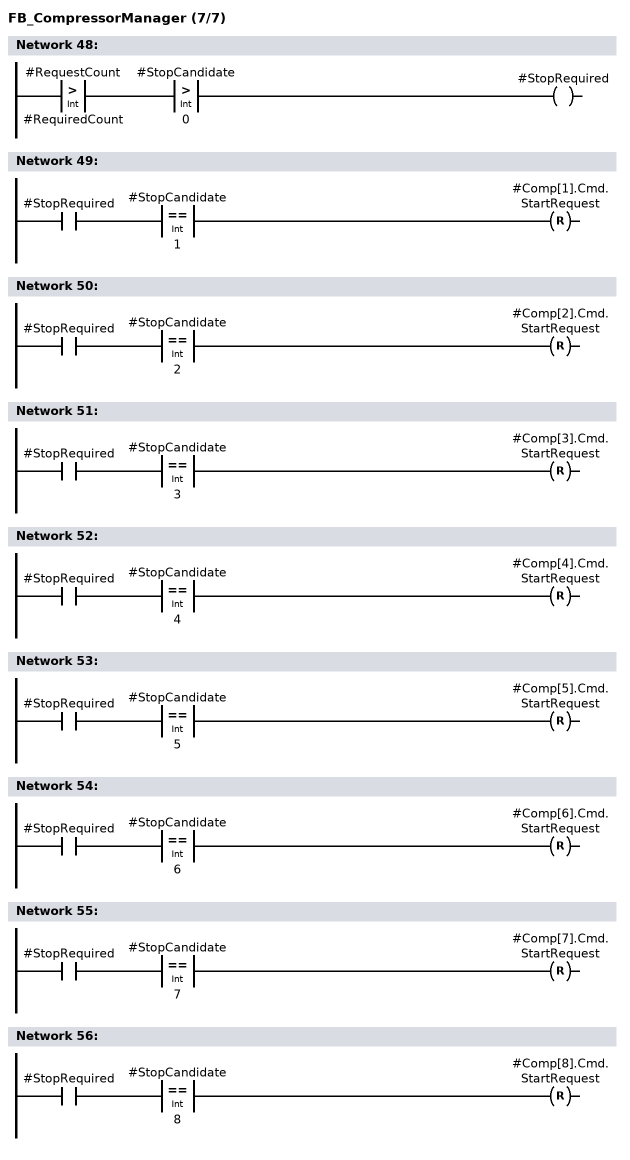
   RUNG wire#powerrail
      { S7_Templates := "SrcType := Int" } GT_Contact(in1 := #RequestCount, in2 := #RequiredCount)
      { S7_Templates := "SrcType := Int" } GT_Contact(in1 := #StopCandidate, in2 := 0)
      Coil( #StopRequired )
   END_RUNG
   // the same network as SCL:
   #StopRequired := (#RequestCount > #RequiredCount) AND (#StopCandidate > 0);
END_REGION

REGION Network 49
   RUNG wire#powerrail
      Contact( #StopRequired )
      { S7_Templates := "SrcType := Int" } EQ_Contact(in1 := #StopCandidate, in2 := 1)
      R_Coil( #Comp[1].Cmd.StartRequest )
   END_RUNG
   // the same network as SCL:
   IF #StopRequired AND (#StopCandidate = 1) THEN #Comp[1].Cmd.StartRequest := FALSE; END_IF;
END_REGION

REGION Network 50
   RUNG wire#powerrail
      Contact( #StopRequired )
      { S7_Templates := "SrcType := Int" } EQ_Contact(in1 := #StopCandidate, in2 := 2)
      R_Coil( #Comp[2].Cmd.StartRequest )
   END_RUNG
   // the same network as SCL:
   IF #StopRequired AND (#StopCandidate = 2) THEN #Comp[2].Cmd.StartRequest := FALSE; END_IF;
END_REGION

REGION Network 51
   RUNG wire#powerrail
      Contact( #StopRequired )
      { S7_Templates := "SrcType := Int" } EQ_Contact(in1 := #StopCandidate, in2 := 3)
      R_Coil( #Comp[3].Cmd.StartRequest )
   END_RUNG
   // the same network as SCL:
   IF #StopRequired AND (#StopCandidate = 3) THEN #Comp[3].Cmd.StartRequest := FALSE; END_IF;
END_REGION

REGION Network 52
   RUNG wire#powerrail
      Contact( #StopRequired )
      { S7_Templates := "SrcType := Int" } EQ_Contact(in1 := #StopCandidate, in2 := 4)
      R_Coil( #Comp[4].Cmd.StartRequest )
   END_RUNG
   // the same network as SCL:
   IF #StopRequired AND (#StopCandidate = 4) THEN #Comp[4].Cmd.StartRequest := FALSE; END_IF;
END_REGION

REGION Network 53
   RUNG wire#powerrail
      Contact( #StopRequired )
      { S7_Templates := "SrcType := Int" } EQ_Contact(in1 := #StopCandidate, in2 := 5)
      R_Coil( #Comp[5].Cmd.StartRequest )
   END_RUNG
   // the same network as SCL:
   IF #StopRequired AND (#StopCandidate = 5) THEN #Comp[5].Cmd.StartRequest := FALSE; END_IF;
END_REGION

REGION Network 54
   RUNG wire#powerrail
      Contact( #StopRequired )
      { S7_Templates := "SrcType := Int" } EQ_Contact(in1 := #StopCandidate, in2 := 6)
      R_Coil( #Comp[6].Cmd.StartRequest )
   END_RUNG
   // the same network as SCL:
   IF #StopRequired AND (#StopCandidate = 6) THEN #Comp[6].Cmd.StartRequest := FALSE; END_IF;
END_REGION

REGION Network 55
   RUNG wire#powerrail
      Contact( #StopRequired )
      { S7_Templates := "SrcType := Int" } EQ_Contact(in1 := #StopCandidate, in2 := 7)
      R_Coil( #Comp[7].Cmd.StartRequest )
   END_RUNG
   // the same network as SCL:
   IF #StopRequired AND (#StopCandidate = 7) THEN #Comp[7].Cmd.StartRequest := FALSE; END_IF;
END_REGION

REGION Network 56
   RUNG wire#powerrail
      Contact( #StopRequired )
      { S7_Templates := "SrcType := Int" } EQ_Contact(in1 := #StopCandidate, in2 := 8)
      R_Coil( #Comp[8].Cmd.StartRequest )
   END_RUNG
   // the same network as SCL:
   IF #StopRequired AND (#StopCandidate = 8) THEN #Comp[8].Cmd.StartRequest := FALSE; END_IF;
END_REGION
END_FUNCTION_BLOCK

FUNCTION_BLOCK "FB_Fan"   // FB3, LAD
{ S7_Optimized_Access := 'TRUE' }
VERSION : 0.1
   VAR_INPUT
      Timing : "UDT_TimingParams";
   END_VAR
   VAR_IN_OUT
      Fan : "UDT_Fan";
   END_VAR
   VAR
      tMinOff : TON_TIME;
      tMinOn : TON_TIME;
      StartLatch : Bool;
      tFeedBack : TON_TIME;
   END_VAR
   VAR_TEMP
      MinOffDone : Bool;
      MinOnDone : Bool;
      StopCondition : Bool;
      FeedbackTimeOut : Bool;
   END_VAR
BEGIN

REGION Network 1
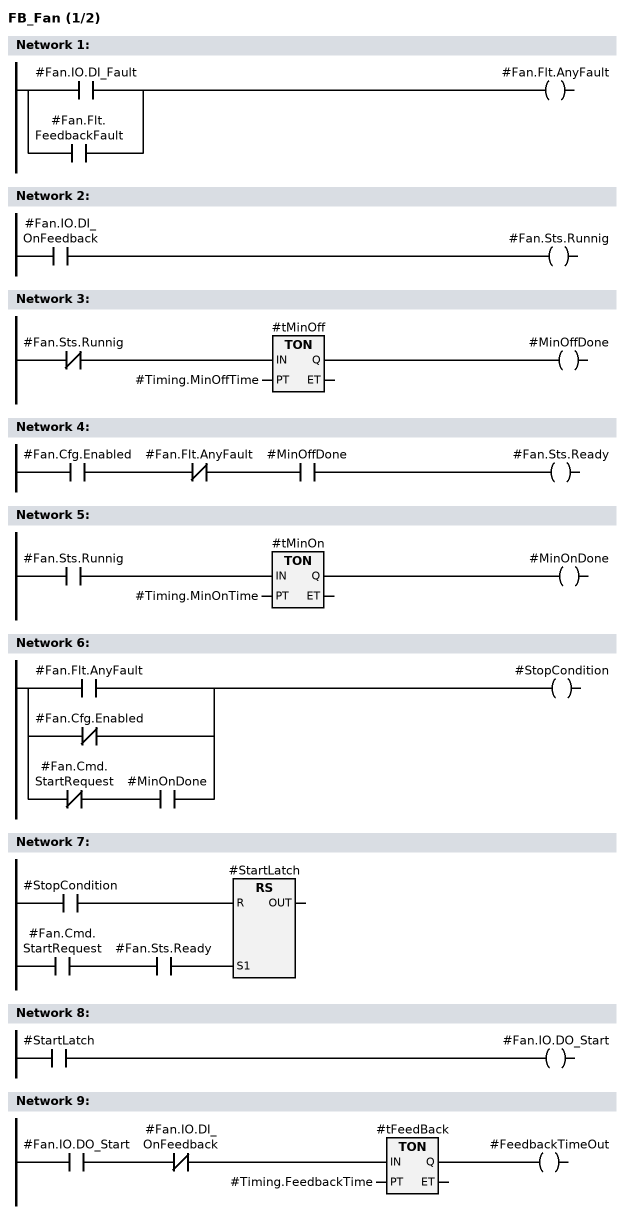
   RUNG wire#powerrail
      Contact( #Fan.IO.DI_Fault )
      wire#w1
      Coil( #Fan.Flt.AnyFault )
   END_RUNG
   RUNG wire#powerrail
      Contact( #Fan.Flt.FeedbackFault )
   END_RUNG wire#w1
   // the same network as SCL:
   #Fan.Flt.AnyFault := #Fan.IO.DI_Fault OR #Fan.Flt.FeedbackFault;
END_REGION

REGION Network 2
   RUNG wire#powerrail
      Contact( #Fan.IO.DI_OnFeedback )
      Coil( #Fan.Sts.Runnig )
   END_RUNG
   // the same network as SCL:
   #Fan.Sts.Runnig := #Fan.IO.DI_OnFeedback;
END_REGION

REGION Network 3
   #tMinOff(IN := NOT #Fan.Sts.Runnig, PT := #Timing.MinOffTime);   // TON
   #MinOffDone := #tMinOff.Q;
END_REGION

REGION Network 4
   RUNG wire#powerrail
      Contact( #Fan.Cfg.Enabled )
      I_Contact( #Fan.Flt.AnyFault )
      Contact( #MinOffDone )
      Coil( #Fan.Sts.Ready )
   END_RUNG
   // the same network as SCL:
   #Fan.Sts.Ready := #Fan.Cfg.Enabled AND NOT #Fan.Flt.AnyFault AND #MinOffDone;
END_REGION

REGION Network 5
   #tMinOn(IN := #Fan.Sts.Runnig, PT := #Timing.MinOnTime);   // TON
   #MinOnDone := #tMinOn.Q;
END_REGION

REGION Network 6
   RUNG wire#powerrail
      Contact( #Fan.Flt.AnyFault )
      wire#w1
      Coil( #StopCondition )
   END_RUNG
   RUNG wire#powerrail
      I_Contact( #Fan.Cfg.Enabled )
   END_RUNG wire#w1
   RUNG wire#powerrail
      I_Contact( #Fan.Cmd.StartRequest )
      Contact( #MinOnDone )
   END_RUNG wire#w1
   // the same network as SCL:
   #StopCondition := #Fan.Flt.AnyFault OR NOT #Fan.Cfg.Enabled OR (NOT #Fan.Cmd.StartRequest AND #MinOnDone);
END_REGION

REGION Network 7
   RUNG wire#powerrail
      Contact( #StopCondition )
      S_RS(operand := #StartLatch, s1 := wire#w1)
   END_RUNG
   RUNG wire#powerrail
      Contact( #Fan.Cmd.StartRequest )
      Contact( #Fan.Sts.Ready )
   END_RUNG wire#w1
   // the same network as SCL:
   IF #StopCondition THEN
       #StartLatch := FALSE;   // RS flip-flop
   END_IF;
   IF #Fan.Cmd.StartRequest AND #Fan.Sts.Ready THEN #StartLatch := TRUE; END_IF;
END_REGION

REGION Network 8
   RUNG wire#powerrail
      Contact( #StartLatch )
      Coil( #Fan.IO.DO_Start )
   END_RUNG
   // the same network as SCL:
   #Fan.IO.DO_Start := #StartLatch;
END_REGION

REGION Network 9
   #tFeedBack(IN := #Fan.IO.DO_Start AND NOT #Fan.IO.DI_OnFeedback, PT := #Timing.FeedbackTime);   // TON
   #FeedbackTimeOut := #tFeedBack.Q;
END_REGION

REGION Network 10
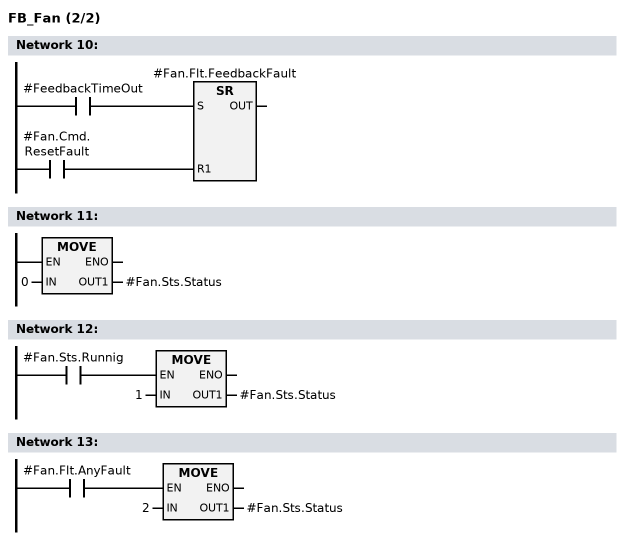
   RUNG wire#powerrail
      Contact( #FeedbackTimeOut )
      S_SR(operand := #Fan.Flt.FeedbackFault, r1 := wire#w1)
   END_RUNG
   RUNG wire#powerrail
      Contact( #Fan.Cmd.ResetFault )
   END_RUNG wire#w1
   // the same network as SCL:
   IF #FeedbackTimeOut THEN
       #Fan.Flt.FeedbackFault := TRUE;   // SR flip-flop
   END_IF;
   IF #Fan.Cmd.ResetFault THEN #Fan.Flt.FeedbackFault := FALSE; END_IF;
END_REGION

REGION Network 11
   RUNG wire#powerrail
      Move(in := 0, out1 => #Fan.Sts.Status)
   END_RUNG
   // the same network as SCL:
   #Fan.Sts.Status := 0;
END_REGION

REGION Network 12
   RUNG wire#powerrail
      Contact( #Fan.Sts.Runnig )
      Move(in := 1, out1 => #Fan.Sts.Status)
   END_RUNG
   // the same network as SCL:
   IF #Fan.Sts.Runnig THEN #Fan.Sts.Status := 1; END_IF;
END_REGION

REGION Network 13
   RUNG wire#powerrail
      Contact( #Fan.Flt.AnyFault )
      Move(in := 2, out1 => #Fan.Sts.Status)
   END_RUNG
   // the same network as SCL:
   IF #Fan.Flt.AnyFault THEN #Fan.Sts.Status := 2; END_IF;
END_REGION
END_FUNCTION_BLOCK

FUNCTION_BLOCK "FB_FanManager"   // FB4, LAD
{ S7_Optimized_Access := 'TRUE' }
VERSION : 0.1
   VAR_INPUT
      Enable : Bool;
      RequiredCount : Int;
   END_VAR
   VAR_OUTPUT
      RunningCount : Int;
      RequestCount : Int;
   END_VAR
   VAR_IN_OUT
      fan : Array[1..12] of "UDT_Fan";
   END_VAR
   VAR_TEMP
      TargetCount : Int;
      StartCandidate : Int;
      StopCandidate : Int;
      StartRequired : Bool;
      StopRequired : Bool;
   END_VAR
BEGIN

REGION Network 1
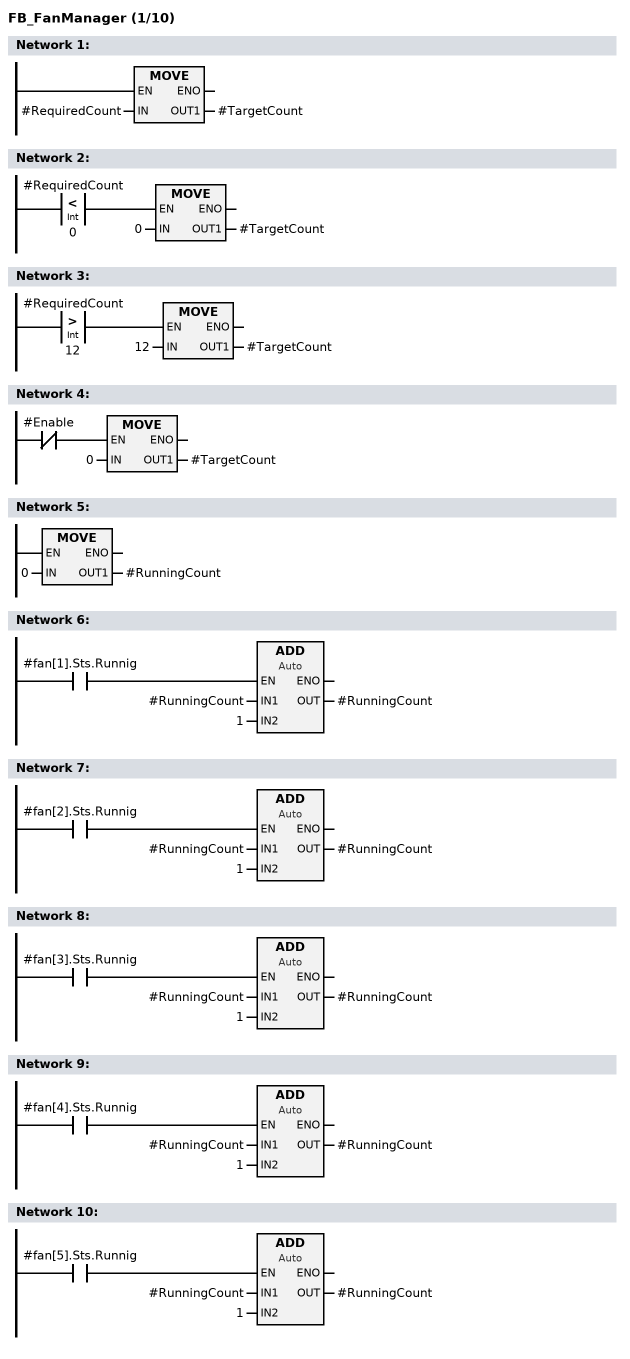
   RUNG wire#powerrail
      Move(in := #RequiredCount, out1 => #TargetCount)
   END_RUNG
   // the same network as SCL:
   #TargetCount := #RequiredCount;
END_REGION

REGION Network 2
   RUNG wire#powerrail
      { S7_Templates := "SrcType := Int" } LT_Contact(in1 := #RequiredCount, in2 := 0)
      Move(in := 0, out1 => #TargetCount)
   END_RUNG
   // the same network as SCL:
   IF #RequiredCount < 0 THEN #TargetCount := 0; END_IF;
END_REGION

REGION Network 3
   RUNG wire#powerrail
      { S7_Templates := "SrcType := Int" } GT_Contact(in1 := #RequiredCount, in2 := 12)
      Move(in := 12, out1 => #TargetCount)
   END_RUNG
   // the same network as SCL:
   IF #RequiredCount > 12 THEN #TargetCount := 12; END_IF;
END_REGION

REGION Network 4
   RUNG wire#powerrail
      I_Contact( #Enable )
      Move(in := 0, out1 => #TargetCount)
   END_RUNG
   // the same network as SCL:
   IF NOT #Enable THEN #TargetCount := 0; END_IF;
END_REGION

REGION Network 5
   RUNG wire#powerrail
      Move(in := 0, out1 => #RunningCount)
   END_RUNG
   // the same network as SCL:
   #RunningCount := 0;
END_REGION

REGION Network 6
   RUNG wire#powerrail
      Contact( #fan[1].Sts.Runnig )
      Add(in1 := #RunningCount, in2 := 1, out => #RunningCount)
   END_RUNG
   // the same network as SCL:
   IF #fan[1].Sts.Runnig THEN #RunningCount := #RunningCount + 1; END_IF;
END_REGION

REGION Network 7
   RUNG wire#powerrail
      Contact( #fan[2].Sts.Runnig )
      Add(in1 := #RunningCount, in2 := 1, out => #RunningCount)
   END_RUNG
   // the same network as SCL:
   IF #fan[2].Sts.Runnig THEN #RunningCount := #RunningCount + 1; END_IF;
END_REGION

REGION Network 8
   RUNG wire#powerrail
      Contact( #fan[3].Sts.Runnig )
      Add(in1 := #RunningCount, in2 := 1, out => #RunningCount)
   END_RUNG
   // the same network as SCL:
   IF #fan[3].Sts.Runnig THEN #RunningCount := #RunningCount + 1; END_IF;
END_REGION

REGION Network 9
   RUNG wire#powerrail
      Contact( #fan[4].Sts.Runnig )
      Add(in1 := #RunningCount, in2 := 1, out => #RunningCount)
   END_RUNG
   // the same network as SCL:
   IF #fan[4].Sts.Runnig THEN #RunningCount := #RunningCount + 1; END_IF;
END_REGION

REGION Network 10
   RUNG wire#powerrail
      Contact( #fan[5].Sts.Runnig )
      Add(in1 := #RunningCount, in2 := 1, out => #RunningCount)
   END_RUNG
   // the same network as SCL:
   IF #fan[5].Sts.Runnig THEN #RunningCount := #RunningCount + 1; END_IF;
END_REGION

REGION Network 11
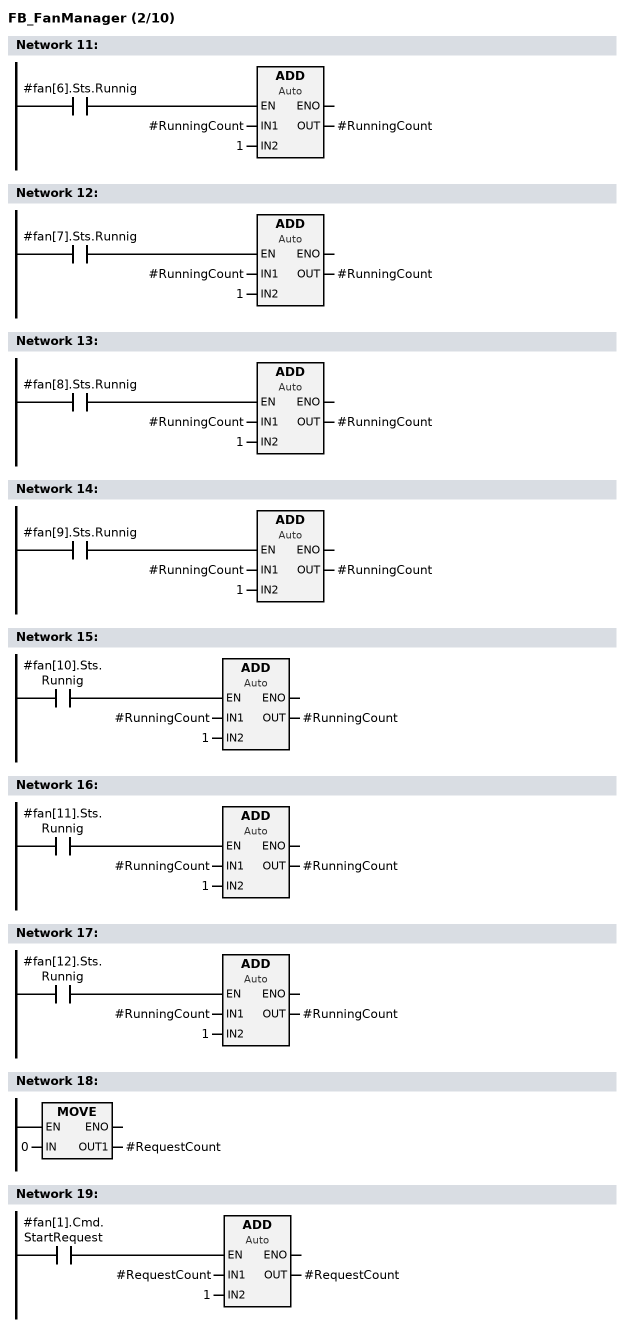
   RUNG wire#powerrail
      Contact( #fan[6].Sts.Runnig )
      Add(in1 := #RunningCount, in2 := 1, out => #RunningCount)
   END_RUNG
   // the same network as SCL:
   IF #fan[6].Sts.Runnig THEN #RunningCount := #RunningCount + 1; END_IF;
END_REGION

REGION Network 12
   RUNG wire#powerrail
      Contact( #fan[7].Sts.Runnig )
      Add(in1 := #RunningCount, in2 := 1, out => #RunningCount)
   END_RUNG
   // the same network as SCL:
   IF #fan[7].Sts.Runnig THEN #RunningCount := #RunningCount + 1; END_IF;
END_REGION

REGION Network 13
   RUNG wire#powerrail
      Contact( #fan[8].Sts.Runnig )
      Add(in1 := #RunningCount, in2 := 1, out => #RunningCount)
   END_RUNG
   // the same network as SCL:
   IF #fan[8].Sts.Runnig THEN #RunningCount := #RunningCount + 1; END_IF;
END_REGION

REGION Network 14
   RUNG wire#powerrail
      Contact( #fan[9].Sts.Runnig )
      Add(in1 := #RunningCount, in2 := 1, out => #RunningCount)
   END_RUNG
   // the same network as SCL:
   IF #fan[9].Sts.Runnig THEN #RunningCount := #RunningCount + 1; END_IF;
END_REGION

REGION Network 15
   RUNG wire#powerrail
      Contact( #fan[10].Sts.Runnig )
      Add(in1 := #RunningCount, in2 := 1, out => #RunningCount)
   END_RUNG
   // the same network as SCL:
   IF #fan[10].Sts.Runnig THEN #RunningCount := #RunningCount + 1; END_IF;
END_REGION

REGION Network 16
   RUNG wire#powerrail
      Contact( #fan[11].Sts.Runnig )
      Add(in1 := #RunningCount, in2 := 1, out => #RunningCount)
   END_RUNG
   // the same network as SCL:
   IF #fan[11].Sts.Runnig THEN #RunningCount := #RunningCount + 1; END_IF;
END_REGION

REGION Network 17
   RUNG wire#powerrail
      Contact( #fan[12].Sts.Runnig )
      Add(in1 := #RunningCount, in2 := 1, out => #RunningCount)
   END_RUNG
   // the same network as SCL:
   IF #fan[12].Sts.Runnig THEN #RunningCount := #RunningCount + 1; END_IF;
END_REGION

REGION Network 18
   RUNG wire#powerrail
      Move(in := 0, out1 => #RequestCount)
   END_RUNG
   // the same network as SCL:
   #RequestCount := 0;
END_REGION

REGION Network 19
   RUNG wire#powerrail
      Contact( #fan[1].Cmd.StartRequest )
      Add(in1 := #RequestCount, in2 := 1, out => #RequestCount)
   END_RUNG
   // the same network as SCL:
   IF #fan[1].Cmd.StartRequest THEN #RequestCount := #RequestCount + 1; END_IF;
END_REGION

REGION Network 20
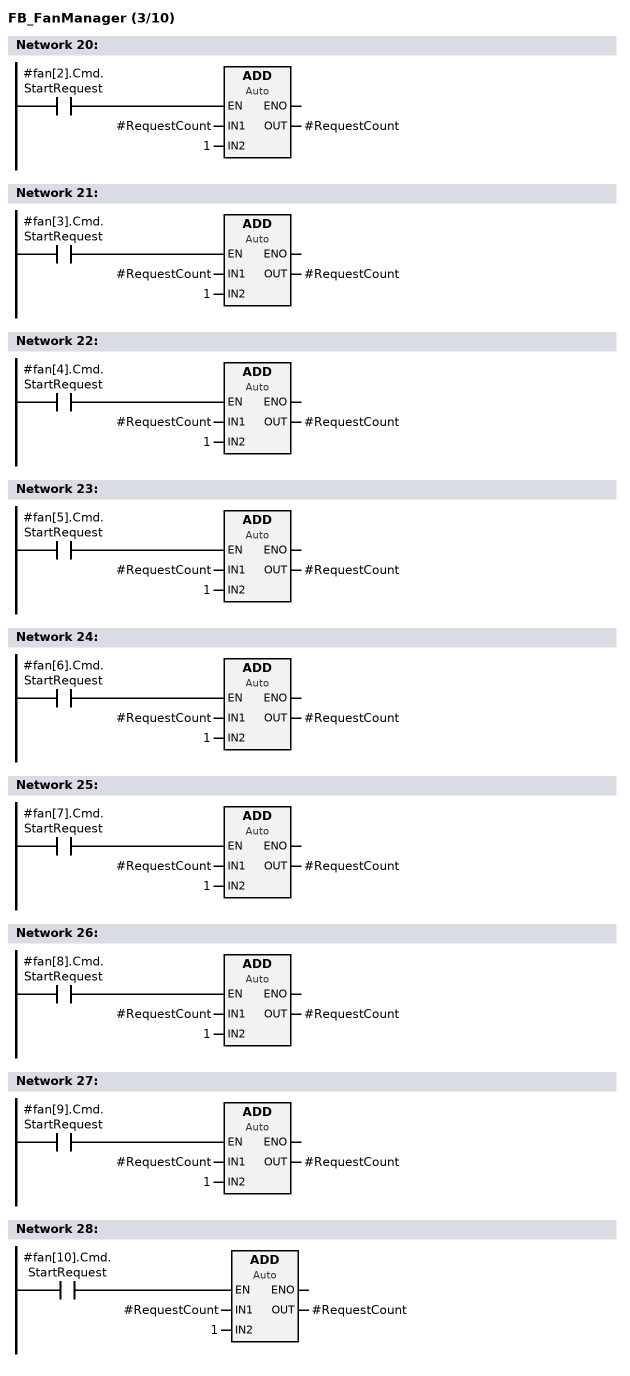
   RUNG wire#powerrail
      Contact( #fan[2].Cmd.StartRequest )
      Add(in1 := #RequestCount, in2 := 1, out => #RequestCount)
   END_RUNG
   // the same network as SCL:
   IF #fan[2].Cmd.StartRequest THEN #RequestCount := #RequestCount + 1; END_IF;
END_REGION

REGION Network 21
   RUNG wire#powerrail
      Contact( #fan[3].Cmd.StartRequest )
      Add(in1 := #RequestCount, in2 := 1, out => #RequestCount)
   END_RUNG
   // the same network as SCL:
   IF #fan[3].Cmd.StartRequest THEN #RequestCount := #RequestCount + 1; END_IF;
END_REGION

REGION Network 22
   RUNG wire#powerrail
      Contact( #fan[4].Cmd.StartRequest )
      Add(in1 := #RequestCount, in2 := 1, out => #RequestCount)
   END_RUNG
   // the same network as SCL:
   IF #fan[4].Cmd.StartRequest THEN #RequestCount := #RequestCount + 1; END_IF;
END_REGION

REGION Network 23
   RUNG wire#powerrail
      Contact( #fan[5].Cmd.StartRequest )
      Add(in1 := #RequestCount, in2 := 1, out => #RequestCount)
   END_RUNG
   // the same network as SCL:
   IF #fan[5].Cmd.StartRequest THEN #RequestCount := #RequestCount + 1; END_IF;
END_REGION

REGION Network 24
   RUNG wire#powerrail
      Contact( #fan[6].Cmd.StartRequest )
      Add(in1 := #RequestCount, in2 := 1, out => #RequestCount)
   END_RUNG
   // the same network as SCL:
   IF #fan[6].Cmd.StartRequest THEN #RequestCount := #RequestCount + 1; END_IF;
END_REGION

REGION Network 25
   RUNG wire#powerrail
      Contact( #fan[7].Cmd.StartRequest )
      Add(in1 := #RequestCount, in2 := 1, out => #RequestCount)
   END_RUNG
   // the same network as SCL:
   IF #fan[7].Cmd.StartRequest THEN #RequestCount := #RequestCount + 1; END_IF;
END_REGION

REGION Network 26
   RUNG wire#powerrail
      Contact( #fan[8].Cmd.StartRequest )
      Add(in1 := #RequestCount, in2 := 1, out => #RequestCount)
   END_RUNG
   // the same network as SCL:
   IF #fan[8].Cmd.StartRequest THEN #RequestCount := #RequestCount + 1; END_IF;
END_REGION

REGION Network 27
   RUNG wire#powerrail
      Contact( #fan[9].Cmd.StartRequest )
      Add(in1 := #RequestCount, in2 := 1, out => #RequestCount)
   END_RUNG
   // the same network as SCL:
   IF #fan[9].Cmd.StartRequest THEN #RequestCount := #RequestCount + 1; END_IF;
END_REGION

REGION Network 28
   RUNG wire#powerrail
      Contact( #fan[10].Cmd.StartRequest )
      Add(in1 := #RequestCount, in2 := 1, out => #RequestCount)
   END_RUNG
   // the same network as SCL:
   IF #fan[10].Cmd.StartRequest THEN #RequestCount := #RequestCount + 1; END_IF;
END_REGION

REGION Network 29
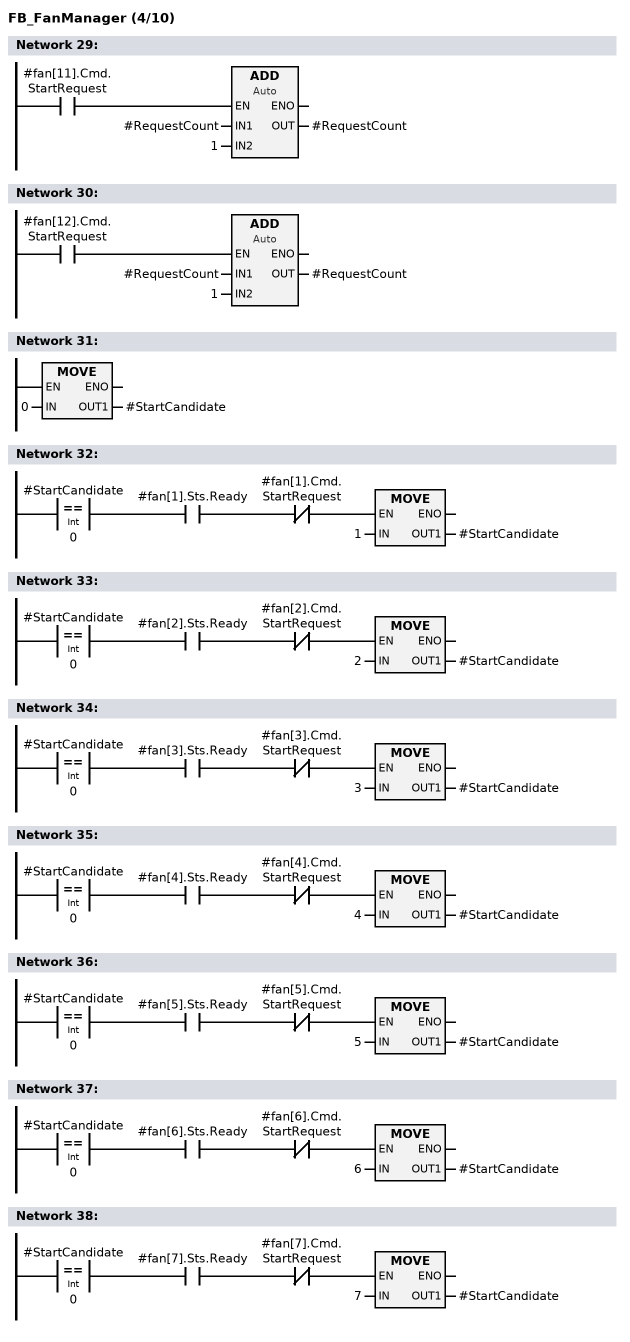
   RUNG wire#powerrail
      Contact( #fan[11].Cmd.StartRequest )
      Add(in1 := #RequestCount, in2 := 1, out => #RequestCount)
   END_RUNG
   // the same network as SCL:
   IF #fan[11].Cmd.StartRequest THEN #RequestCount := #RequestCount + 1; END_IF;
END_REGION

REGION Network 30
   RUNG wire#powerrail
      Contact( #fan[12].Cmd.StartRequest )
      Add(in1 := #RequestCount, in2 := 1, out => #RequestCount)
   END_RUNG
   // the same network as SCL:
   IF #fan[12].Cmd.StartRequest THEN #RequestCount := #RequestCount + 1; END_IF;
END_REGION

REGION Network 31
   RUNG wire#powerrail
      Move(in := 0, out1 => #StartCandidate)
   END_RUNG
   // the same network as SCL:
   #StartCandidate := 0;
END_REGION

REGION Network 32
   RUNG wire#powerrail
      { S7_Templates := "SrcType := Int" } EQ_Contact(in1 := #StartCandidate, in2 := 0)
      Contact( #fan[1].Sts.Ready )
      I_Contact( #fan[1].Cmd.StartRequest )
      Move(in := 1, out1 => #StartCandidate)
   END_RUNG
   // the same network as SCL:
   IF (#StartCandidate = 0) AND #fan[1].Sts.Ready AND NOT #fan[1].Cmd.StartRequest THEN
       #StartCandidate := 1;
   END_IF;
END_REGION

REGION Network 33
   RUNG wire#powerrail
      { S7_Templates := "SrcType := Int" } EQ_Contact(in1 := #StartCandidate, in2 := 0)
      Contact( #fan[2].Sts.Ready )
      I_Contact( #fan[2].Cmd.StartRequest )
      Move(in := 2, out1 => #StartCandidate)
   END_RUNG
   // the same network as SCL:
   IF (#StartCandidate = 0) AND #fan[2].Sts.Ready AND NOT #fan[2].Cmd.StartRequest THEN
       #StartCandidate := 2;
   END_IF;
END_REGION

REGION Network 34
   RUNG wire#powerrail
      { S7_Templates := "SrcType := Int" } EQ_Contact(in1 := #StartCandidate, in2 := 0)
      Contact( #fan[3].Sts.Ready )
      I_Contact( #fan[3].Cmd.StartRequest )
      Move(in := 3, out1 => #StartCandidate)
   END_RUNG
   // the same network as SCL:
   IF (#StartCandidate = 0) AND #fan[3].Sts.Ready AND NOT #fan[3].Cmd.StartRequest THEN
       #StartCandidate := 3;
   END_IF;
END_REGION

REGION Network 35
   RUNG wire#powerrail
      { S7_Templates := "SrcType := Int" } EQ_Contact(in1 := #StartCandidate, in2 := 0)
      Contact( #fan[4].Sts.Ready )
      I_Contact( #fan[4].Cmd.StartRequest )
      Move(in := 4, out1 => #StartCandidate)
   END_RUNG
   // the same network as SCL:
   IF (#StartCandidate = 0) AND #fan[4].Sts.Ready AND NOT #fan[4].Cmd.StartRequest THEN
       #StartCandidate := 4;
   END_IF;
END_REGION

REGION Network 36
   RUNG wire#powerrail
      { S7_Templates := "SrcType := Int" } EQ_Contact(in1 := #StartCandidate, in2 := 0)
      Contact( #fan[5].Sts.Ready )
      I_Contact( #fan[5].Cmd.StartRequest )
      Move(in := 5, out1 => #StartCandidate)
   END_RUNG
   // the same network as SCL:
   IF (#StartCandidate = 0) AND #fan[5].Sts.Ready AND NOT #fan[5].Cmd.StartRequest THEN
       #StartCandidate := 5;
   END_IF;
END_REGION

REGION Network 37
   RUNG wire#powerrail
      { S7_Templates := "SrcType := Int" } EQ_Contact(in1 := #StartCandidate, in2 := 0)
      Contact( #fan[6].Sts.Ready )
      I_Contact( #fan[6].Cmd.StartRequest )
      Move(in := 6, out1 => #StartCandidate)
   END_RUNG
   // the same network as SCL:
   IF (#StartCandidate = 0) AND #fan[6].Sts.Ready AND NOT #fan[6].Cmd.StartRequest THEN
       #StartCandidate := 6;
   END_IF;
END_REGION

REGION Network 38
   RUNG wire#powerrail
      { S7_Templates := "SrcType := Int" } EQ_Contact(in1 := #StartCandidate, in2 := 0)
      Contact( #fan[7].Sts.Ready )
      I_Contact( #fan[7].Cmd.StartRequest )
      Move(in := 7, out1 => #StartCandidate)
   END_RUNG
   // the same network as SCL:
   IF (#StartCandidate = 0) AND #fan[7].Sts.Ready AND NOT #fan[7].Cmd.StartRequest THEN
       #StartCandidate := 7;
   END_IF;
END_REGION

REGION Network 39
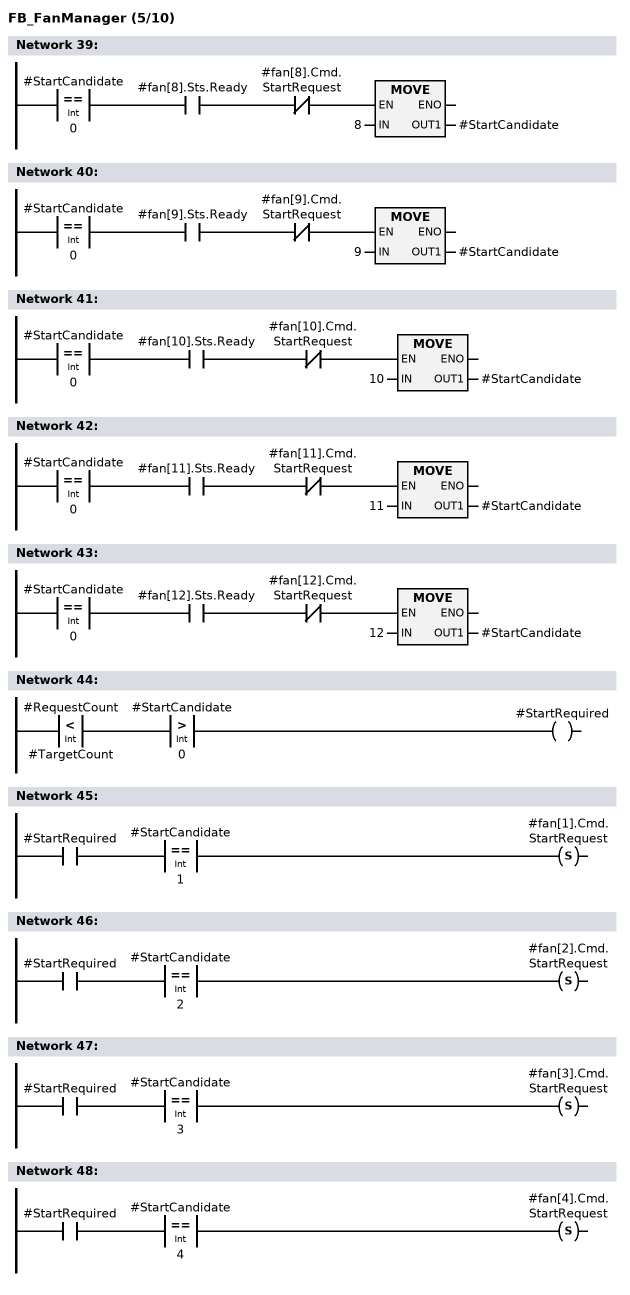
   RUNG wire#powerrail
      { S7_Templates := "SrcType := Int" } EQ_Contact(in1 := #StartCandidate, in2 := 0)
      Contact( #fan[8].Sts.Ready )
      I_Contact( #fan[8].Cmd.StartRequest )
      Move(in := 8, out1 => #StartCandidate)
   END_RUNG
   // the same network as SCL:
   IF (#StartCandidate = 0) AND #fan[8].Sts.Ready AND NOT #fan[8].Cmd.StartRequest THEN
       #StartCandidate := 8;
   END_IF;
END_REGION

REGION Network 40
   RUNG wire#powerrail
      { S7_Templates := "SrcType := Int" } EQ_Contact(in1 := #StartCandidate, in2 := 0)
      Contact( #fan[9].Sts.Ready )
      I_Contact( #fan[9].Cmd.StartRequest )
      Move(in := 9, out1 => #StartCandidate)
   END_RUNG
   // the same network as SCL:
   IF (#StartCandidate = 0) AND #fan[9].Sts.Ready AND NOT #fan[9].Cmd.StartRequest THEN
       #StartCandidate := 9;
   END_IF;
END_REGION

REGION Network 41
   RUNG wire#powerrail
      { S7_Templates := "SrcType := Int" } EQ_Contact(in1 := #StartCandidate, in2 := 0)
      Contact( #fan[10].Sts.Ready )
      I_Contact( #fan[10].Cmd.StartRequest )
      Move(in := 10, out1 => #StartCandidate)
   END_RUNG
   // the same network as SCL:
   IF (#StartCandidate = 0) AND #fan[10].Sts.Ready AND NOT #fan[10].Cmd.StartRequest THEN
       #StartCandidate := 10;
   END_IF;
END_REGION

REGION Network 42
   RUNG wire#powerrail
      { S7_Templates := "SrcType := Int" } EQ_Contact(in1 := #StartCandidate, in2 := 0)
      Contact( #fan[11].Sts.Ready )
      I_Contact( #fan[11].Cmd.StartRequest )
      Move(in := 11, out1 => #StartCandidate)
   END_RUNG
   // the same network as SCL:
   IF (#StartCandidate = 0) AND #fan[11].Sts.Ready AND NOT #fan[11].Cmd.StartRequest THEN
       #StartCandidate := 11;
   END_IF;
END_REGION

REGION Network 43
   RUNG wire#powerrail
      { S7_Templates := "SrcType := Int" } EQ_Contact(in1 := #StartCandidate, in2 := 0)
      Contact( #fan[12].Sts.Ready )
      I_Contact( #fan[12].Cmd.StartRequest )
      Move(in := 12, out1 => #StartCandidate)
   END_RUNG
   // the same network as SCL:
   IF (#StartCandidate = 0) AND #fan[12].Sts.Ready AND NOT #fan[12].Cmd.StartRequest THEN
       #StartCandidate := 12;
   END_IF;
END_REGION

REGION Network 44
   RUNG wire#powerrail
      { S7_Templates := "SrcType := Int" } LT_Contact(in1 := #RequestCount, in2 := #TargetCount)
      { S7_Templates := "SrcType := Int" } GT_Contact(in1 := #StartCandidate, in2 := 0)
      Coil( #StartRequired )
   END_RUNG
   // the same network as SCL:
   #StartRequired := (#RequestCount < #TargetCount) AND (#StartCandidate > 0);
END_REGION

REGION Network 45
   RUNG wire#powerrail
      Contact( #StartRequired )
      { S7_Templates := "SrcType := Int" } EQ_Contact(in1 := #StartCandidate, in2 := 1)
      S_Coil( #fan[1].Cmd.StartRequest )
   END_RUNG
   // the same network as SCL:
   IF #StartRequired AND (#StartCandidate = 1) THEN #fan[1].Cmd.StartRequest := TRUE; END_IF;
END_REGION

REGION Network 46
   RUNG wire#powerrail
      Contact( #StartRequired )
      { S7_Templates := "SrcType := Int" } EQ_Contact(in1 := #StartCandidate, in2 := 2)
      S_Coil( #fan[2].Cmd.StartRequest )
   END_RUNG
   // the same network as SCL:
   IF #StartRequired AND (#StartCandidate = 2) THEN #fan[2].Cmd.StartRequest := TRUE; END_IF;
END_REGION

REGION Network 47
   RUNG wire#powerrail
      Contact( #StartRequired )
      { S7_Templates := "SrcType := Int" } EQ_Contact(in1 := #StartCandidate, in2 := 3)
      S_Coil( #fan[3].Cmd.StartRequest )
   END_RUNG
   // the same network as SCL:
   IF #StartRequired AND (#StartCandidate = 3) THEN #fan[3].Cmd.StartRequest := TRUE; END_IF;
END_REGION

REGION Network 48
   RUNG wire#powerrail
      Contact( #StartRequired )
      { S7_Templates := "SrcType := Int" } EQ_Contact(in1 := #StartCandidate, in2 := 4)
      S_Coil( #fan[4].Cmd.StartRequest )
   END_RUNG
   // the same network as SCL:
   IF #StartRequired AND (#StartCandidate = 4) THEN #fan[4].Cmd.StartRequest := TRUE; END_IF;
END_REGION

REGION Network 49
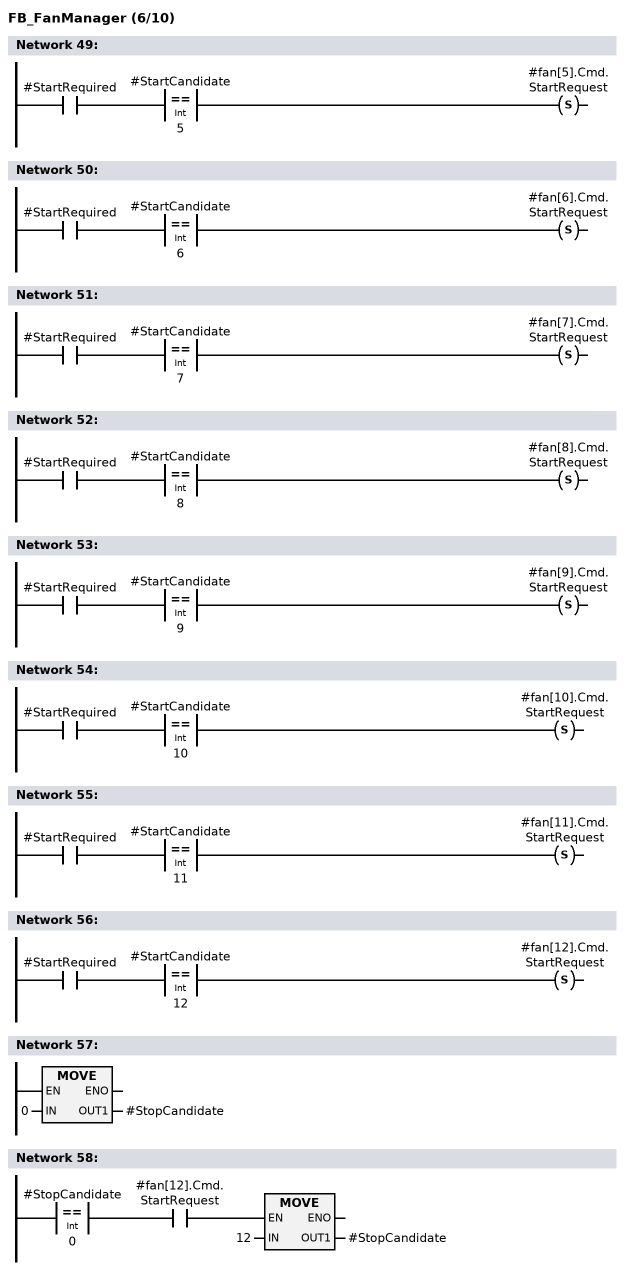
   RUNG wire#powerrail
      Contact( #StartRequired )
      { S7_Templates := "SrcType := Int" } EQ_Contact(in1 := #StartCandidate, in2 := 5)
      S_Coil( #fan[5].Cmd.StartRequest )
   END_RUNG
   // the same network as SCL:
   IF #StartRequired AND (#StartCandidate = 5) THEN #fan[5].Cmd.StartRequest := TRUE; END_IF;
END_REGION

REGION Network 50
   RUNG wire#powerrail
      Contact( #StartRequired )
      { S7_Templates := "SrcType := Int" } EQ_Contact(in1 := #StartCandidate, in2 := 6)
      S_Coil( #fan[6].Cmd.StartRequest )
   END_RUNG
   // the same network as SCL:
   IF #StartRequired AND (#StartCandidate = 6) THEN #fan[6].Cmd.StartRequest := TRUE; END_IF;
END_REGION

REGION Network 51
   RUNG wire#powerrail
      Contact( #StartRequired )
      { S7_Templates := "SrcType := Int" } EQ_Contact(in1 := #StartCandidate, in2 := 7)
      S_Coil( #fan[7].Cmd.StartRequest )
   END_RUNG
   // the same network as SCL:
   IF #StartRequired AND (#StartCandidate = 7) THEN #fan[7].Cmd.StartRequest := TRUE; END_IF;
END_REGION

REGION Network 52
   RUNG wire#powerrail
      Contact( #StartRequired )
      { S7_Templates := "SrcType := Int" } EQ_Contact(in1 := #StartCandidate, in2 := 8)
      S_Coil( #fan[8].Cmd.StartRequest )
   END_RUNG
   // the same network as SCL:
   IF #StartRequired AND (#StartCandidate = 8) THEN #fan[8].Cmd.StartRequest := TRUE; END_IF;
END_REGION

REGION Network 53
   RUNG wire#powerrail
      Contact( #StartRequired )
      { S7_Templates := "SrcType := Int" } EQ_Contact(in1 := #StartCandidate, in2 := 9)
      S_Coil( #fan[9].Cmd.StartRequest )
   END_RUNG
   // the same network as SCL:
   IF #StartRequired AND (#StartCandidate = 9) THEN #fan[9].Cmd.StartRequest := TRUE; END_IF;
END_REGION

REGION Network 54
   RUNG wire#powerrail
      Contact( #StartRequired )
      { S7_Templates := "SrcType := Int" } EQ_Contact(in1 := #StartCandidate, in2 := 10)
      S_Coil( #fan[10].Cmd.StartRequest )
   END_RUNG
   // the same network as SCL:
   IF #StartRequired AND (#StartCandidate = 10) THEN #fan[10].Cmd.StartRequest := TRUE; END_IF;
END_REGION

REGION Network 55
   RUNG wire#powerrail
      Contact( #StartRequired )
      { S7_Templates := "SrcType := Int" } EQ_Contact(in1 := #StartCandidate, in2 := 11)
      S_Coil( #fan[11].Cmd.StartRequest )
   END_RUNG
   // the same network as SCL:
   IF #StartRequired AND (#StartCandidate = 11) THEN #fan[11].Cmd.StartRequest := TRUE; END_IF;
END_REGION

REGION Network 56
   RUNG wire#powerrail
      Contact( #StartRequired )
      { S7_Templates := "SrcType := Int" } EQ_Contact(in1 := #StartCandidate, in2 := 12)
      S_Coil( #fan[12].Cmd.StartRequest )
   END_RUNG
   // the same network as SCL:
   IF #StartRequired AND (#StartCandidate = 12) THEN #fan[12].Cmd.StartRequest := TRUE; END_IF;
END_REGION

REGION Network 57
   RUNG wire#powerrail
      Move(in := 0, out1 => #StopCandidate)
   END_RUNG
   // the same network as SCL:
   #StopCandidate := 0;
END_REGION

REGION Network 58
   RUNG wire#powerrail
      { S7_Templates := "SrcType := Int" } EQ_Contact(in1 := #StopCandidate, in2 := 0)
      Contact( #fan[12].Cmd.StartRequest )
      Move(in := 12, out1 => #StopCandidate)
   END_RUNG
   // the same network as SCL:
   IF (#StopCandidate = 0) AND #fan[12].Cmd.StartRequest THEN #StopCandidate := 12; END_IF;
END_REGION

REGION Network 59
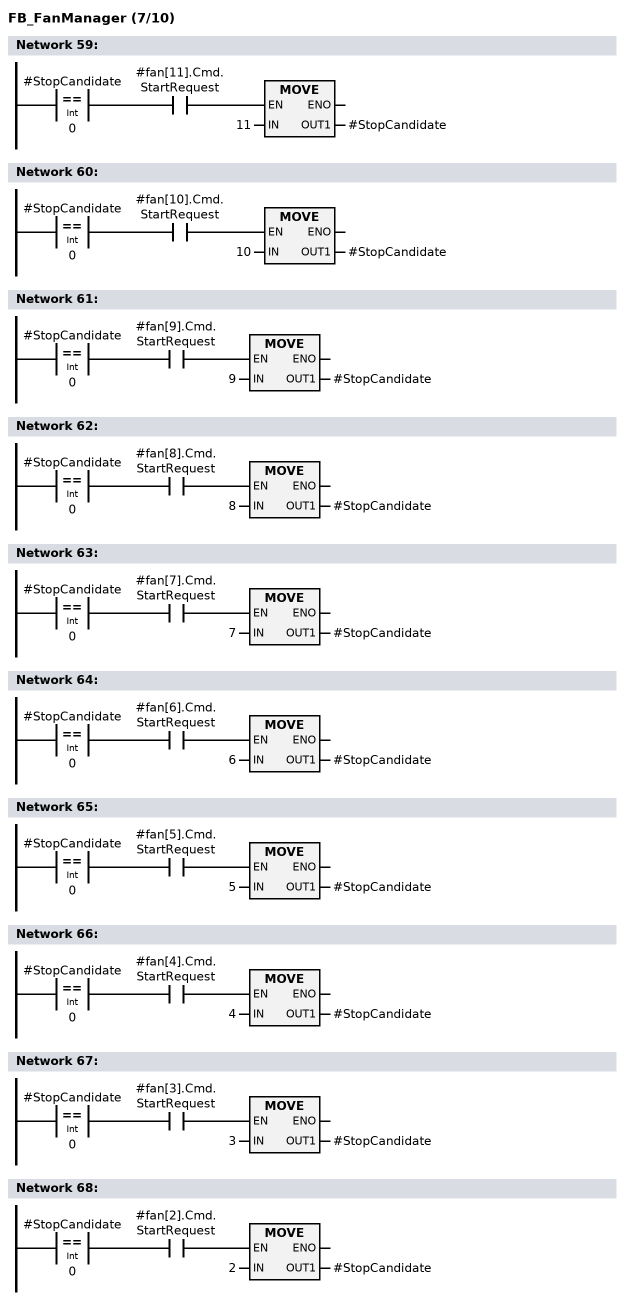
   RUNG wire#powerrail
      { S7_Templates := "SrcType := Int" } EQ_Contact(in1 := #StopCandidate, in2 := 0)
      Contact( #fan[11].Cmd.StartRequest )
      Move(in := 11, out1 => #StopCandidate)
   END_RUNG
   // the same network as SCL:
   IF (#StopCandidate = 0) AND #fan[11].Cmd.StartRequest THEN #StopCandidate := 11; END_IF;
END_REGION

REGION Network 60
   RUNG wire#powerrail
      { S7_Templates := "SrcType := Int" } EQ_Contact(in1 := #StopCandidate, in2 := 0)
      Contact( #fan[10].Cmd.StartRequest )
      Move(in := 10, out1 => #StopCandidate)
   END_RUNG
   // the same network as SCL:
   IF (#StopCandidate = 0) AND #fan[10].Cmd.StartRequest THEN #StopCandidate := 10; END_IF;
END_REGION

REGION Network 61
   RUNG wire#powerrail
      { S7_Templates := "SrcType := Int" } EQ_Contact(in1 := #StopCandidate, in2 := 0)
      Contact( #fan[9].Cmd.StartRequest )
      Move(in := 9, out1 => #StopCandidate)
   END_RUNG
   // the same network as SCL:
   IF (#StopCandidate = 0) AND #fan[9].Cmd.StartRequest THEN #StopCandidate := 9; END_IF;
END_REGION

REGION Network 62
   RUNG wire#powerrail
      { S7_Templates := "SrcType := Int" } EQ_Contact(in1 := #StopCandidate, in2 := 0)
      Contact( #fan[8].Cmd.StartRequest )
      Move(in := 8, out1 => #StopCandidate)
   END_RUNG
   // the same network as SCL:
   IF (#StopCandidate = 0) AND #fan[8].Cmd.StartRequest THEN #StopCandidate := 8; END_IF;
END_REGION

REGION Network 63
   RUNG wire#powerrail
      { S7_Templates := "SrcType := Int" } EQ_Contact(in1 := #StopCandidate, in2 := 0)
      Contact( #fan[7].Cmd.StartRequest )
      Move(in := 7, out1 => #StopCandidate)
   END_RUNG
   // the same network as SCL:
   IF (#StopCandidate = 0) AND #fan[7].Cmd.StartRequest THEN #StopCandidate := 7; END_IF;
END_REGION

REGION Network 64
   RUNG wire#powerrail
      { S7_Templates := "SrcType := Int" } EQ_Contact(in1 := #StopCandidate, in2 := 0)
      Contact( #fan[6].Cmd.StartRequest )
      Move(in := 6, out1 => #StopCandidate)
   END_RUNG
   // the same network as SCL:
   IF (#StopCandidate = 0) AND #fan[6].Cmd.StartRequest THEN #StopCandidate := 6; END_IF;
END_REGION

REGION Network 65
   RUNG wire#powerrail
      { S7_Templates := "SrcType := Int" } EQ_Contact(in1 := #StopCandidate, in2 := 0)
      Contact( #fan[5].Cmd.StartRequest )
      Move(in := 5, out1 => #StopCandidate)
   END_RUNG
   // the same network as SCL:
   IF (#StopCandidate = 0) AND #fan[5].Cmd.StartRequest THEN #StopCandidate := 5; END_IF;
END_REGION

REGION Network 66
   RUNG wire#powerrail
      { S7_Templates := "SrcType := Int" } EQ_Contact(in1 := #StopCandidate, in2 := 0)
      Contact( #fan[4].Cmd.StartRequest )
      Move(in := 4, out1 => #StopCandidate)
   END_RUNG
   // the same network as SCL:
   IF (#StopCandidate = 0) AND #fan[4].Cmd.StartRequest THEN #StopCandidate := 4; END_IF;
END_REGION

REGION Network 67
   RUNG wire#powerrail
      { S7_Templates := "SrcType := Int" } EQ_Contact(in1 := #StopCandidate, in2 := 0)
      Contact( #fan[3].Cmd.StartRequest )
      Move(in := 3, out1 => #StopCandidate)
   END_RUNG
   // the same network as SCL:
   IF (#StopCandidate = 0) AND #fan[3].Cmd.StartRequest THEN #StopCandidate := 3; END_IF;
END_REGION

REGION Network 68
   RUNG wire#powerrail
      { S7_Templates := "SrcType := Int" } EQ_Contact(in1 := #StopCandidate, in2 := 0)
      Contact( #fan[2].Cmd.StartRequest )
      Move(in := 2, out1 => #StopCandidate)
   END_RUNG
   // the same network as SCL:
   IF (#StopCandidate = 0) AND #fan[2].Cmd.StartRequest THEN #StopCandidate := 2; END_IF;
END_REGION

REGION Network 69
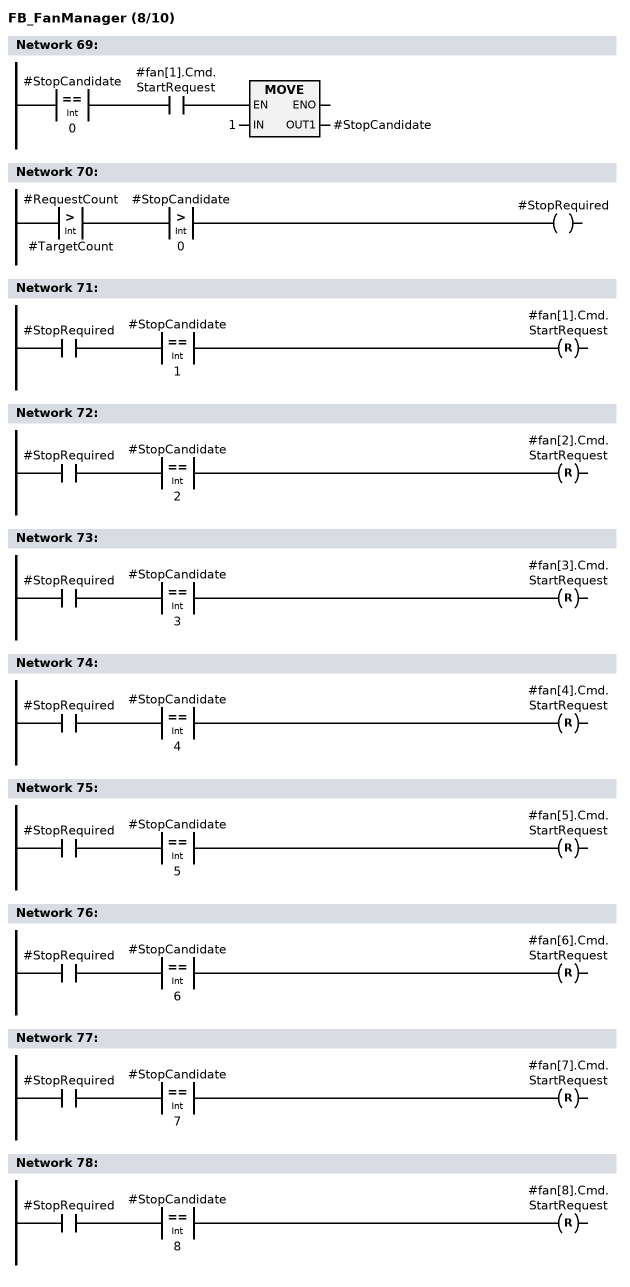
   RUNG wire#powerrail
      { S7_Templates := "SrcType := Int" } EQ_Contact(in1 := #StopCandidate, in2 := 0)
      Contact( #fan[1].Cmd.StartRequest )
      Move(in := 1, out1 => #StopCandidate)
   END_RUNG
   // the same network as SCL:
   IF (#StopCandidate = 0) AND #fan[1].Cmd.StartRequest THEN #StopCandidate := 1; END_IF;
END_REGION

REGION Network 70
   RUNG wire#powerrail
      { S7_Templates := "SrcType := Int" } GT_Contact(in1 := #RequestCount, in2 := #TargetCount)
      { S7_Templates := "SrcType := Int" } GT_Contact(in1 := #StopCandidate, in2 := 0)
      Coil( #StopRequired )
   END_RUNG
   // the same network as SCL:
   #StopRequired := (#RequestCount > #TargetCount) AND (#StopCandidate > 0);
END_REGION

REGION Network 71
   RUNG wire#powerrail
      Contact( #StopRequired )
      { S7_Templates := "SrcType := Int" } EQ_Contact(in1 := #StopCandidate, in2 := 1)
      R_Coil( #fan[1].Cmd.StartRequest )
   END_RUNG
   // the same network as SCL:
   IF #StopRequired AND (#StopCandidate = 1) THEN #fan[1].Cmd.StartRequest := FALSE; END_IF;
END_REGION

REGION Network 72
   RUNG wire#powerrail
      Contact( #StopRequired )
      { S7_Templates := "SrcType := Int" } EQ_Contact(in1 := #StopCandidate, in2 := 2)
      R_Coil( #fan[2].Cmd.StartRequest )
   END_RUNG
   // the same network as SCL:
   IF #StopRequired AND (#StopCandidate = 2) THEN #fan[2].Cmd.StartRequest := FALSE; END_IF;
END_REGION

REGION Network 73
   RUNG wire#powerrail
      Contact( #StopRequired )
      { S7_Templates := "SrcType := Int" } EQ_Contact(in1 := #StopCandidate, in2 := 3)
      R_Coil( #fan[3].Cmd.StartRequest )
   END_RUNG
   // the same network as SCL:
   IF #StopRequired AND (#StopCandidate = 3) THEN #fan[3].Cmd.StartRequest := FALSE; END_IF;
END_REGION

REGION Network 74
   RUNG wire#powerrail
      Contact( #StopRequired )
      { S7_Templates := "SrcType := Int" } EQ_Contact(in1 := #StopCandidate, in2 := 4)
      R_Coil( #fan[4].Cmd.StartRequest )
   END_RUNG
   // the same network as SCL:
   IF #StopRequired AND (#StopCandidate = 4) THEN #fan[4].Cmd.StartRequest := FALSE; END_IF;
END_REGION

REGION Network 75
   RUNG wire#powerrail
      Contact( #StopRequired )
      { S7_Templates := "SrcType := Int" } EQ_Contact(in1 := #StopCandidate, in2 := 5)
      R_Coil( #fan[5].Cmd.StartRequest )
   END_RUNG
   // the same network as SCL:
   IF #StopRequired AND (#StopCandidate = 5) THEN #fan[5].Cmd.StartRequest := FALSE; END_IF;
END_REGION

REGION Network 76
   RUNG wire#powerrail
      Contact( #StopRequired )
      { S7_Templates := "SrcType := Int" } EQ_Contact(in1 := #StopCandidate, in2 := 6)
      R_Coil( #fan[6].Cmd.StartRequest )
   END_RUNG
   // the same network as SCL:
   IF #StopRequired AND (#StopCandidate = 6) THEN #fan[6].Cmd.StartRequest := FALSE; END_IF;
END_REGION

REGION Network 77
   RUNG wire#powerrail
      Contact( #StopRequired )
      { S7_Templates := "SrcType := Int" } EQ_Contact(in1 := #StopCandidate, in2 := 7)
      R_Coil( #fan[7].Cmd.StartRequest )
   END_RUNG
   // the same network as SCL:
   IF #StopRequired AND (#StopCandidate = 7) THEN #fan[7].Cmd.StartRequest := FALSE; END_IF;
END_REGION

REGION Network 78
   RUNG wire#powerrail
      Contact( #StopRequired )
      { S7_Templates := "SrcType := Int" } EQ_Contact(in1 := #StopCandidate, in2 := 8)
      R_Coil( #fan[8].Cmd.StartRequest )
   END_RUNG
   // the same network as SCL:
   IF #StopRequired AND (#StopCandidate = 8) THEN #fan[8].Cmd.StartRequest := FALSE; END_IF;
END_REGION

REGION Network 79
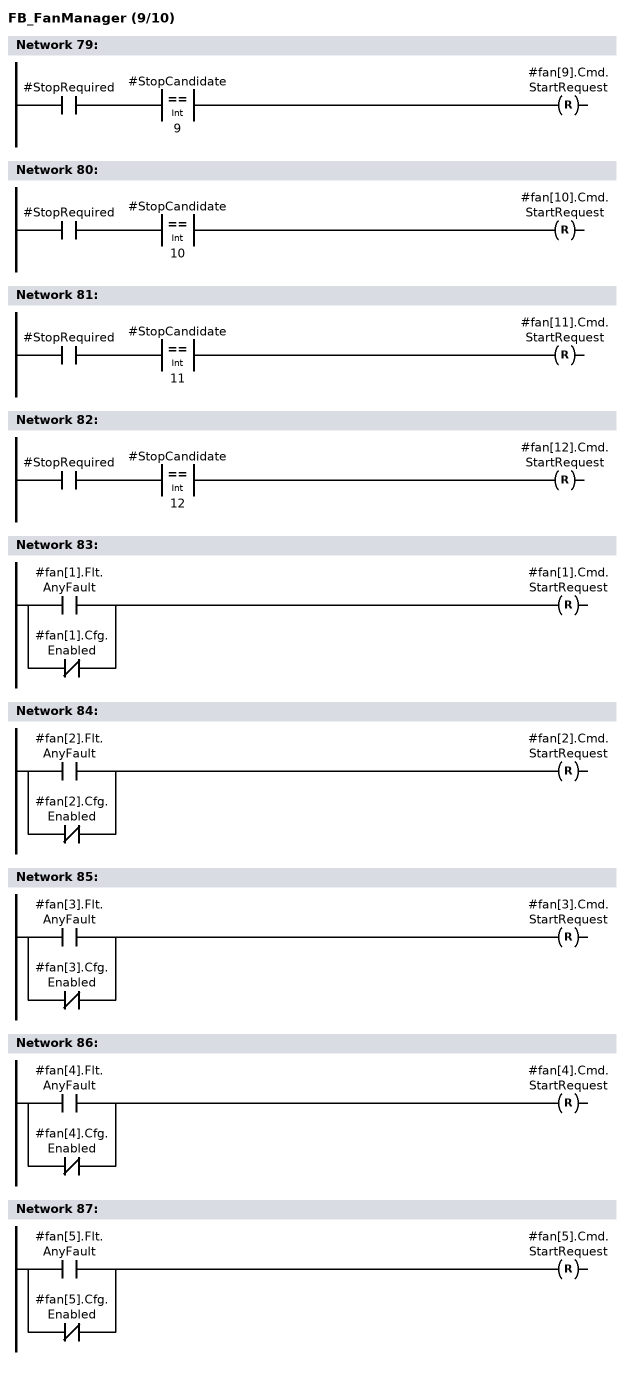
   RUNG wire#powerrail
      Contact( #StopRequired )
      { S7_Templates := "SrcType := Int" } EQ_Contact(in1 := #StopCandidate, in2 := 9)
      R_Coil( #fan[9].Cmd.StartRequest )
   END_RUNG
   // the same network as SCL:
   IF #StopRequired AND (#StopCandidate = 9) THEN #fan[9].Cmd.StartRequest := FALSE; END_IF;
END_REGION

REGION Network 80
   RUNG wire#powerrail
      Contact( #StopRequired )
      { S7_Templates := "SrcType := Int" } EQ_Contact(in1 := #StopCandidate, in2 := 10)
      R_Coil( #fan[10].Cmd.StartRequest )
   END_RUNG
   // the same network as SCL:
   IF #StopRequired AND (#StopCandidate = 10) THEN #fan[10].Cmd.StartRequest := FALSE; END_IF;
END_REGION

REGION Network 81
   RUNG wire#powerrail
      Contact( #StopRequired )
      { S7_Templates := "SrcType := Int" } EQ_Contact(in1 := #StopCandidate, in2 := 11)
      R_Coil( #fan[11].Cmd.StartRequest )
   END_RUNG
   // the same network as SCL:
   IF #StopRequired AND (#StopCandidate = 11) THEN #fan[11].Cmd.StartRequest := FALSE; END_IF;
END_REGION

REGION Network 82
   RUNG wire#powerrail
      Contact( #StopRequired )
      { S7_Templates := "SrcType := Int" } EQ_Contact(in1 := #StopCandidate, in2 := 12)
      R_Coil( #fan[12].Cmd.StartRequest )
   END_RUNG
   // the same network as SCL:
   IF #StopRequired AND (#StopCandidate = 12) THEN #fan[12].Cmd.StartRequest := FALSE; END_IF;
END_REGION

REGION Network 83
   RUNG wire#powerrail
      Contact( #fan[1].Flt.AnyFault )
      wire#w1
      R_Coil( #fan[1].Cmd.StartRequest )
   END_RUNG
   RUNG wire#powerrail
      I_Contact( #fan[1].Cfg.Enabled )
   END_RUNG wire#w1
   // the same network as SCL:
   IF #fan[1].Flt.AnyFault OR NOT #fan[1].Cfg.Enabled THEN #fan[1].Cmd.StartRequest := FALSE; END_IF;
END_REGION

REGION Network 84
   RUNG wire#powerrail
      Contact( #fan[2].Flt.AnyFault )
      wire#w1
      R_Coil( #fan[2].Cmd.StartRequest )
   END_RUNG
   RUNG wire#powerrail
      I_Contact( #fan[2].Cfg.Enabled )
   END_RUNG wire#w1
   // the same network as SCL:
   IF #fan[2].Flt.AnyFault OR NOT #fan[2].Cfg.Enabled THEN #fan[2].Cmd.StartRequest := FALSE; END_IF;
END_REGION

REGION Network 85
   RUNG wire#powerrail
      Contact( #fan[3].Flt.AnyFault )
      wire#w1
      R_Coil( #fan[3].Cmd.StartRequest )
   END_RUNG
   RUNG wire#powerrail
      I_Contact( #fan[3].Cfg.Enabled )
   END_RUNG wire#w1
   // the same network as SCL:
   IF #fan[3].Flt.AnyFault OR NOT #fan[3].Cfg.Enabled THEN #fan[3].Cmd.StartRequest := FALSE; END_IF;
END_REGION

REGION Network 86
   RUNG wire#powerrail
      Contact( #fan[4].Flt.AnyFault )
      wire#w1
      R_Coil( #fan[4].Cmd.StartRequest )
   END_RUNG
   RUNG wire#powerrail
      I_Contact( #fan[4].Cfg.Enabled )
   END_RUNG wire#w1
   // the same network as SCL:
   IF #fan[4].Flt.AnyFault OR NOT #fan[4].Cfg.Enabled THEN #fan[4].Cmd.StartRequest := FALSE; END_IF;
END_REGION

REGION Network 87
   RUNG wire#powerrail
      Contact( #fan[5].Flt.AnyFault )
      wire#w1
      R_Coil( #fan[5].Cmd.StartRequest )
   END_RUNG
   RUNG wire#powerrail
      I_Contact( #fan[5].Cfg.Enabled )
   END_RUNG wire#w1
   // the same network as SCL:
   IF #fan[5].Flt.AnyFault OR NOT #fan[5].Cfg.Enabled THEN #fan[5].Cmd.StartRequest := FALSE; END_IF;
END_REGION

REGION Network 88
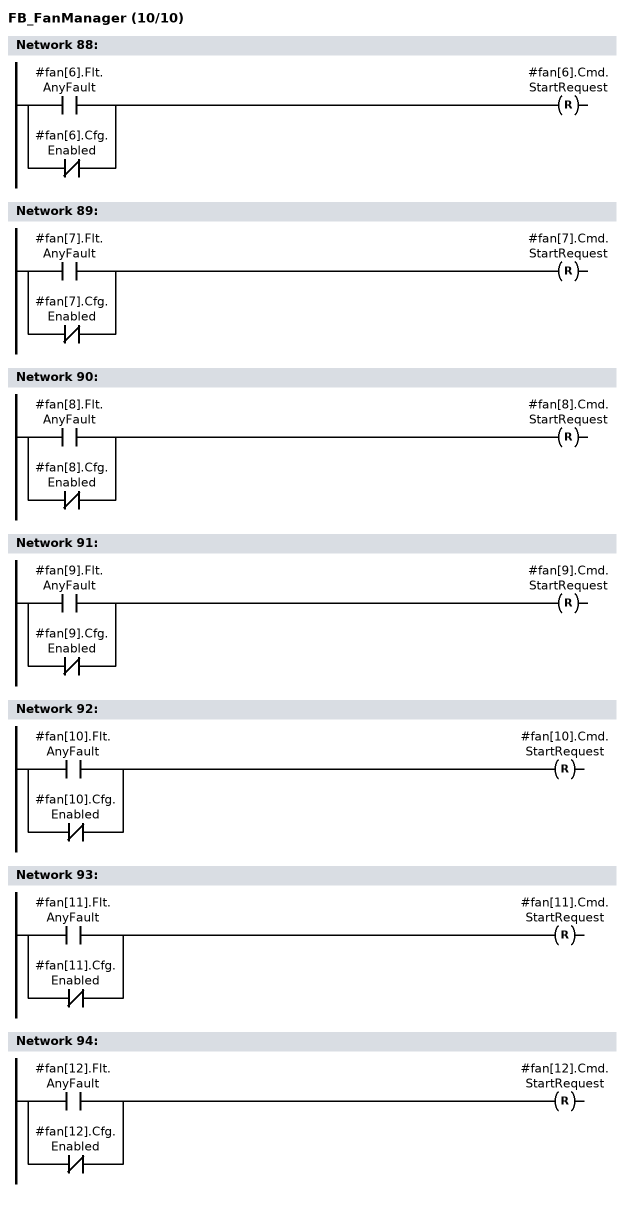
   RUNG wire#powerrail
      Contact( #fan[6].Flt.AnyFault )
      wire#w1
      R_Coil( #fan[6].Cmd.StartRequest )
   END_RUNG
   RUNG wire#powerrail
      I_Contact( #fan[6].Cfg.Enabled )
   END_RUNG wire#w1
   // the same network as SCL:
   IF #fan[6].Flt.AnyFault OR NOT #fan[6].Cfg.Enabled THEN #fan[6].Cmd.StartRequest := FALSE; END_IF;
END_REGION

REGION Network 89
   RUNG wire#powerrail
      Contact( #fan[7].Flt.AnyFault )
      wire#w1
      R_Coil( #fan[7].Cmd.StartRequest )
   END_RUNG
   RUNG wire#powerrail
      I_Contact( #fan[7].Cfg.Enabled )
   END_RUNG wire#w1
   // the same network as SCL:
   IF #fan[7].Flt.AnyFault OR NOT #fan[7].Cfg.Enabled THEN #fan[7].Cmd.StartRequest := FALSE; END_IF;
END_REGION

REGION Network 90
   RUNG wire#powerrail
      Contact( #fan[8].Flt.AnyFault )
      wire#w1
      R_Coil( #fan[8].Cmd.StartRequest )
   END_RUNG
   RUNG wire#powerrail
      I_Contact( #fan[8].Cfg.Enabled )
   END_RUNG wire#w1
   // the same network as SCL:
   IF #fan[8].Flt.AnyFault OR NOT #fan[8].Cfg.Enabled THEN #fan[8].Cmd.StartRequest := FALSE; END_IF;
END_REGION

REGION Network 91
   RUNG wire#powerrail
      Contact( #fan[9].Flt.AnyFault )
      wire#w1
      R_Coil( #fan[9].Cmd.StartRequest )
   END_RUNG
   RUNG wire#powerrail
      I_Contact( #fan[9].Cfg.Enabled )
   END_RUNG wire#w1
   // the same network as SCL:
   IF #fan[9].Flt.AnyFault OR NOT #fan[9].Cfg.Enabled THEN #fan[9].Cmd.StartRequest := FALSE; END_IF;
END_REGION

REGION Network 92
   RUNG wire#powerrail
      Contact( #fan[10].Flt.AnyFault )
      wire#w1
      R_Coil( #fan[10].Cmd.StartRequest )
   END_RUNG
   RUNG wire#powerrail
      I_Contact( #fan[10].Cfg.Enabled )
   END_RUNG wire#w1
   // the same network as SCL:
   IF #fan[10].Flt.AnyFault OR NOT #fan[10].Cfg.Enabled THEN #fan[10].Cmd.StartRequest := FALSE; END_IF;
END_REGION

REGION Network 93
   RUNG wire#powerrail
      Contact( #fan[11].Flt.AnyFault )
      wire#w1
      R_Coil( #fan[11].Cmd.StartRequest )
   END_RUNG
   RUNG wire#powerrail
      I_Contact( #fan[11].Cfg.Enabled )
   END_RUNG wire#w1
   // the same network as SCL:
   IF #fan[11].Flt.AnyFault OR NOT #fan[11].Cfg.Enabled THEN #fan[11].Cmd.StartRequest := FALSE; END_IF;
END_REGION

REGION Network 94
   RUNG wire#powerrail
      Contact( #fan[12].Flt.AnyFault )
      wire#w1
      R_Coil( #fan[12].Cmd.StartRequest )
   END_RUNG
   RUNG wire#powerrail
      I_Contact( #fan[12].Cfg.Enabled )
   END_RUNG wire#w1
   // the same network as SCL:
   IF #fan[12].Flt.AnyFault OR NOT #fan[12].Cfg.Enabled THEN #fan[12].Cmd.StartRequest := FALSE; END_IF;
END_REGION
END_FUNCTION_BLOCK

// folder: 02_utilities

FUNCTION "FC_CalcPercent" : Void   // FC1, LAD
{ S7_Optimized_Access := 'TRUE' }
VERSION : 0.1
   VAR_INPUT
      totalequipment : Int;
      RunningCount : Int;
   END_VAR
   VAR_OUTPUT
      Percent : Real;
   END_VAR
   VAR_TEMP
      RunningReal : Real;
      TotalReal : Real;
      Ratio : Real;
   END_VAR
BEGIN

REGION Network 1
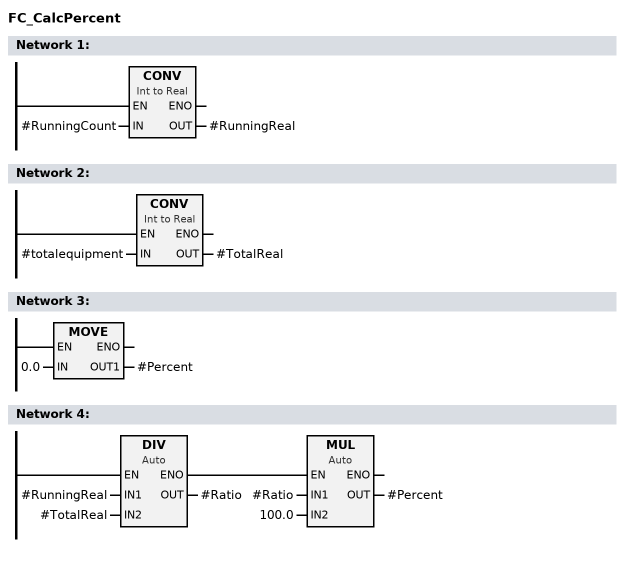
   RUNG wire#powerrail
      { S7_Templates := "[SrcType := Int, DestType := Real]" } Convert(in := #RunningCount, out => #RunningReal)
   END_RUNG
   // the same network as SCL:
   #RunningReal := INT_TO_REAL(#RunningCount);
END_REGION

REGION Network 2
   RUNG wire#powerrail
      { S7_Templates := "[SrcType := Int, DestType := Real]" } Convert(in := #totalequipment, out => #TotalReal)
   END_RUNG
   // the same network as SCL:
   #TotalReal := INT_TO_REAL(#totalequipment);
END_REGION

REGION Network 3
   RUNG wire#powerrail
      Move(in := 0.0, out1 => #Percent)
   END_RUNG
   // the same network as SCL:
   #Percent := 0.0;
END_REGION

REGION Network 4
   RUNG wire#powerrail
      Div(in1 := #RunningReal, in2 := #TotalReal, out => #Ratio)
      Mul(in1 := #Ratio, in2 := 100.0, out => #Percent)
   END_RUNG
   // the same network as SCL:
   #Ratio := #RunningReal / #TotalReal;
   #Percent := #Ratio * 100.0;
END_REGION
END_FUNCTION

FUNCTION "FC_ReadInputs" : Void   // FC2, LAD
{ S7_Optimized_Access := 'TRUE' }
VERSION : 0.1
BEGIN

REGION Network 1
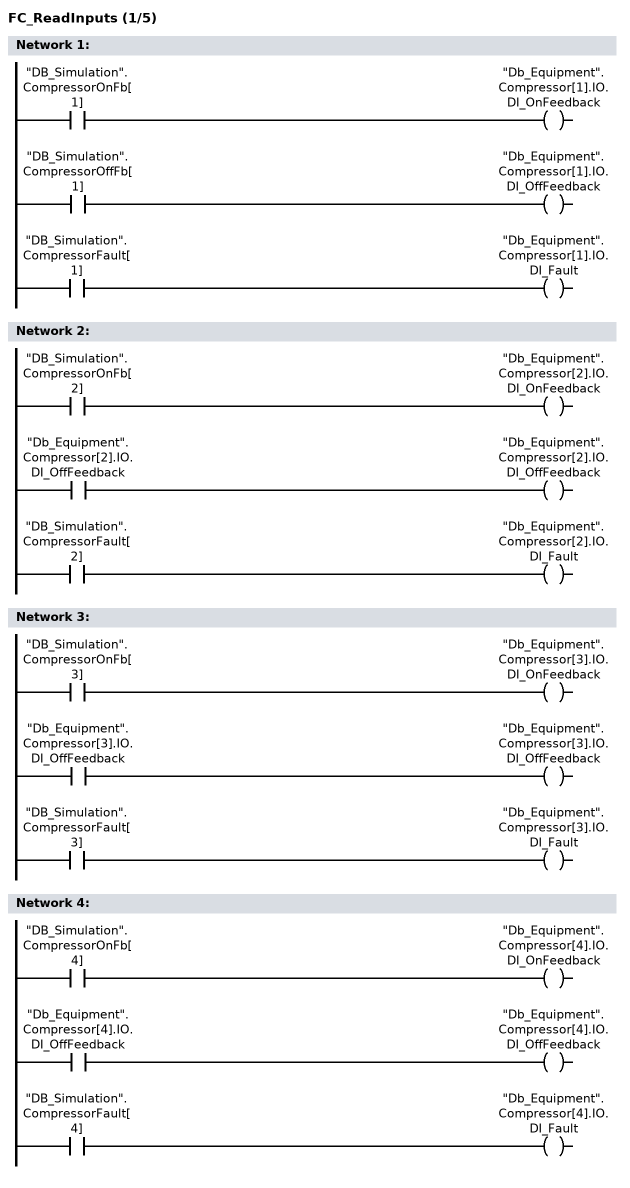
   RUNG wire#powerrail
      Contact( "DB_Simulation".CompressorOnFb[1] )
      Coil( "Db_Equipment".Compressor[1].IO.DI_OnFeedback )
   END_RUNG
   RUNG wire#powerrail
      Contact( "DB_Simulation".CompressorOffFb[1] )
      Coil( "Db_Equipment".Compressor[1].IO.DI_OffFeedback )
   END_RUNG
   RUNG wire#powerrail
      Contact( "DB_Simulation".CompressorFault[1] )
      Coil( "Db_Equipment".Compressor[1].IO.DI_Fault )
   END_RUNG
   // the same network as SCL:
   "Db_Equipment".Compressor[1].IO.DI_OnFeedback := "DB_Simulation".CompressorOnFb[1];
   "Db_Equipment".Compressor[1].IO.DI_OffFeedback := "DB_Simulation".CompressorOffFb[1];
   "Db_Equipment".Compressor[1].IO.DI_Fault := "DB_Simulation".CompressorFault[1];
END_REGION

REGION Network 2
   RUNG wire#powerrail
      Contact( "DB_Simulation".CompressorOnFb[2] )
      Coil( "Db_Equipment".Compressor[2].IO.DI_OnFeedback )
   END_RUNG
   RUNG wire#powerrail
      Contact( "Db_Equipment".Compressor[2].IO.DI_OffFeedback )
      Coil( "Db_Equipment".Compressor[2].IO.DI_OffFeedback )
   END_RUNG
   RUNG wire#powerrail
      Contact( "DB_Simulation".CompressorFault[2] )
      Coil( "Db_Equipment".Compressor[2].IO.DI_Fault )
   END_RUNG
   // the same network as SCL:
   "Db_Equipment".Compressor[2].IO.DI_OnFeedback := "DB_Simulation".CompressorOnFb[2];
   "Db_Equipment".Compressor[2].IO.DI_OffFeedback := "Db_Equipment".Compressor[2].IO.DI_OffFeedback;
   "Db_Equipment".Compressor[2].IO.DI_Fault := "DB_Simulation".CompressorFault[2];
END_REGION

REGION Network 3
   RUNG wire#powerrail
      Contact( "DB_Simulation".CompressorOnFb[3] )
      Coil( "Db_Equipment".Compressor[3].IO.DI_OnFeedback )
   END_RUNG
   RUNG wire#powerrail
      Contact( "Db_Equipment".Compressor[3].IO.DI_OffFeedback )
      Coil( "Db_Equipment".Compressor[3].IO.DI_OffFeedback )
   END_RUNG
   RUNG wire#powerrail
      Contact( "DB_Simulation".CompressorFault[3] )
      Coil( "Db_Equipment".Compressor[3].IO.DI_Fault )
   END_RUNG
   // the same network as SCL:
   "Db_Equipment".Compressor[3].IO.DI_OnFeedback := "DB_Simulation".CompressorOnFb[3];
   "Db_Equipment".Compressor[3].IO.DI_OffFeedback := "Db_Equipment".Compressor[3].IO.DI_OffFeedback;
   "Db_Equipment".Compressor[3].IO.DI_Fault := "DB_Simulation".CompressorFault[3];
END_REGION

REGION Network 4
   RUNG wire#powerrail
      Contact( "DB_Simulation".CompressorOnFb[4] )
      Coil( "Db_Equipment".Compressor[4].IO.DI_OnFeedback )
   END_RUNG
   RUNG wire#powerrail
      Contact( "Db_Equipment".Compressor[4].IO.DI_OffFeedback )
      Coil( "Db_Equipment".Compressor[4].IO.DI_OffFeedback )
   END_RUNG
   RUNG wire#powerrail
      Contact( "DB_Simulation".CompressorFault[4] )
      Coil( "Db_Equipment".Compressor[4].IO.DI_Fault )
   END_RUNG
   // the same network as SCL:
   "Db_Equipment".Compressor[4].IO.DI_OnFeedback := "DB_Simulation".CompressorOnFb[4];
   "Db_Equipment".Compressor[4].IO.DI_OffFeedback := "Db_Equipment".Compressor[4].IO.DI_OffFeedback;
   "Db_Equipment".Compressor[4].IO.DI_Fault := "DB_Simulation".CompressorFault[4];
END_REGION

REGION Network 5
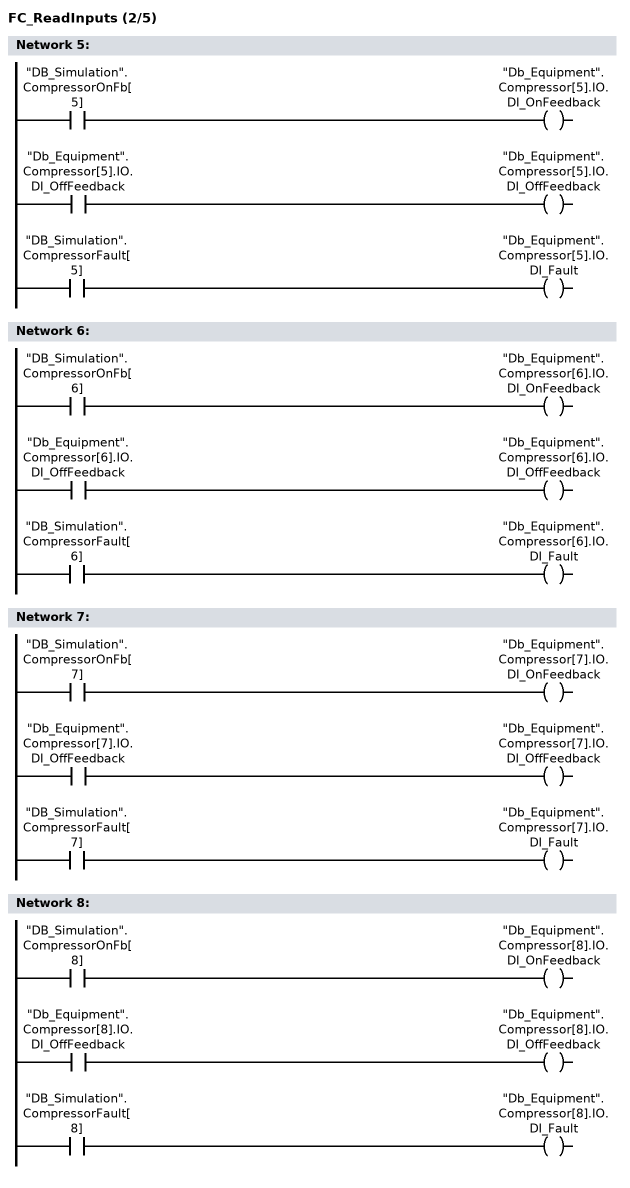
   RUNG wire#powerrail
      Contact( "DB_Simulation".CompressorOnFb[5] )
      Coil( "Db_Equipment".Compressor[5].IO.DI_OnFeedback )
   END_RUNG
   RUNG wire#powerrail
      Contact( "Db_Equipment".Compressor[5].IO.DI_OffFeedback )
      Coil( "Db_Equipment".Compressor[5].IO.DI_OffFeedback )
   END_RUNG
   RUNG wire#powerrail
      Contact( "DB_Simulation".CompressorFault[5] )
      Coil( "Db_Equipment".Compressor[5].IO.DI_Fault )
   END_RUNG
   // the same network as SCL:
   "Db_Equipment".Compressor[5].IO.DI_OnFeedback := "DB_Simulation".CompressorOnFb[5];
   "Db_Equipment".Compressor[5].IO.DI_OffFeedback := "Db_Equipment".Compressor[5].IO.DI_OffFeedback;
   "Db_Equipment".Compressor[5].IO.DI_Fault := "DB_Simulation".CompressorFault[5];
END_REGION

REGION Network 6
   RUNG wire#powerrail
      Contact( "DB_Simulation".CompressorOnFb[6] )
      Coil( "Db_Equipment".Compressor[6].IO.DI_OnFeedback )
   END_RUNG
   RUNG wire#powerrail
      Contact( "Db_Equipment".Compressor[6].IO.DI_OffFeedback )
      Coil( "Db_Equipment".Compressor[6].IO.DI_OffFeedback )
   END_RUNG
   RUNG wire#powerrail
      Contact( "DB_Simulation".CompressorFault[6] )
      Coil( "Db_Equipment".Compressor[6].IO.DI_Fault )
   END_RUNG
   // the same network as SCL:
   "Db_Equipment".Compressor[6].IO.DI_OnFeedback := "DB_Simulation".CompressorOnFb[6];
   "Db_Equipment".Compressor[6].IO.DI_OffFeedback := "Db_Equipment".Compressor[6].IO.DI_OffFeedback;
   "Db_Equipment".Compressor[6].IO.DI_Fault := "DB_Simulation".CompressorFault[6];
END_REGION

REGION Network 7
   RUNG wire#powerrail
      Contact( "DB_Simulation".CompressorOnFb[7] )
      Coil( "Db_Equipment".Compressor[7].IO.DI_OnFeedback )
   END_RUNG
   RUNG wire#powerrail
      Contact( "Db_Equipment".Compressor[7].IO.DI_OffFeedback )
      Coil( "Db_Equipment".Compressor[7].IO.DI_OffFeedback )
   END_RUNG
   RUNG wire#powerrail
      Contact( "DB_Simulation".CompressorFault[7] )
      Coil( "Db_Equipment".Compressor[7].IO.DI_Fault )
   END_RUNG
   // the same network as SCL:
   "Db_Equipment".Compressor[7].IO.DI_OnFeedback := "DB_Simulation".CompressorOnFb[7];
   "Db_Equipment".Compressor[7].IO.DI_OffFeedback := "Db_Equipment".Compressor[7].IO.DI_OffFeedback;
   "Db_Equipment".Compressor[7].IO.DI_Fault := "DB_Simulation".CompressorFault[7];
END_REGION

REGION Network 8
   RUNG wire#powerrail
      Contact( "DB_Simulation".CompressorOnFb[8] )
      Coil( "Db_Equipment".Compressor[8].IO.DI_OnFeedback )
   END_RUNG
   RUNG wire#powerrail
      Contact( "Db_Equipment".Compressor[8].IO.DI_OffFeedback )
      Coil( "Db_Equipment".Compressor[8].IO.DI_OffFeedback )
   END_RUNG
   RUNG wire#powerrail
      Contact( "DB_Simulation".CompressorFault[8] )
      Coil( "Db_Equipment".Compressor[8].IO.DI_Fault )
   END_RUNG
   // the same network as SCL:
   "Db_Equipment".Compressor[8].IO.DI_OnFeedback := "DB_Simulation".CompressorOnFb[8];
   "Db_Equipment".Compressor[8].IO.DI_OffFeedback := "Db_Equipment".Compressor[8].IO.DI_OffFeedback;
   "Db_Equipment".Compressor[8].IO.DI_Fault := "DB_Simulation".CompressorFault[8];
END_REGION

REGION Network 9
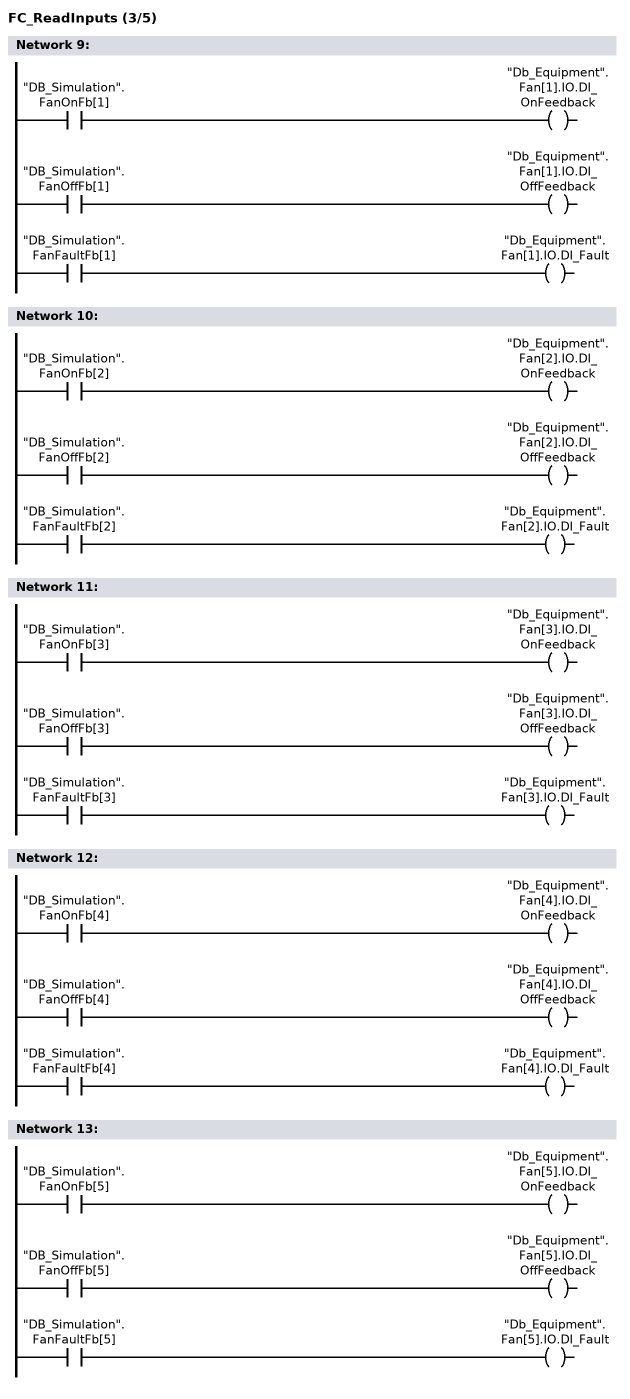
   RUNG wire#powerrail
      Contact( "DB_Simulation".FanOnFb[1] )
      Coil( "Db_Equipment".Fan[1].IO.DI_OnFeedback )
   END_RUNG
   RUNG wire#powerrail
      Contact( "DB_Simulation".FanOffFb[1] )
      Coil( "Db_Equipment".Fan[1].IO.DI_OffFeedback )
   END_RUNG
   RUNG wire#powerrail
      Contact( "DB_Simulation".FanFaultFb[1] )
      Coil( "Db_Equipment".Fan[1].IO.DI_Fault )
   END_RUNG
   // the same network as SCL:
   "Db_Equipment".Fan[1].IO.DI_OnFeedback := "DB_Simulation".FanOnFb[1];
   "Db_Equipment".Fan[1].IO.DI_OffFeedback := "DB_Simulation".FanOffFb[1];
   "Db_Equipment".Fan[1].IO.DI_Fault := "DB_Simulation".FanFaultFb[1];
END_REGION

REGION Network 10
   RUNG wire#powerrail
      Contact( "DB_Simulation".FanOnFb[2] )
      Coil( "Db_Equipment".Fan[2].IO.DI_OnFeedback )
   END_RUNG
   RUNG wire#powerrail
      Contact( "DB_Simulation".FanOffFb[2] )
      Coil( "Db_Equipment".Fan[2].IO.DI_OffFeedback )
   END_RUNG
   RUNG wire#powerrail
      Contact( "DB_Simulation".FanFaultFb[2] )
      Coil( "Db_Equipment".Fan[2].IO.DI_Fault )
   END_RUNG
   // the same network as SCL:
   "Db_Equipment".Fan[2].IO.DI_OnFeedback := "DB_Simulation".FanOnFb[2];
   "Db_Equipment".Fan[2].IO.DI_OffFeedback := "DB_Simulation".FanOffFb[2];
   "Db_Equipment".Fan[2].IO.DI_Fault := "DB_Simulation".FanFaultFb[2];
END_REGION

REGION Network 11
   RUNG wire#powerrail
      Contact( "DB_Simulation".FanOnFb[3] )
      Coil( "Db_Equipment".Fan[3].IO.DI_OnFeedback )
   END_RUNG
   RUNG wire#powerrail
      Contact( "DB_Simulation".FanOffFb[3] )
      Coil( "Db_Equipment".Fan[3].IO.DI_OffFeedback )
   END_RUNG
   RUNG wire#powerrail
      Contact( "DB_Simulation".FanFaultFb[3] )
      Coil( "Db_Equipment".Fan[3].IO.DI_Fault )
   END_RUNG
   // the same network as SCL:
   "Db_Equipment".Fan[3].IO.DI_OnFeedback := "DB_Simulation".FanOnFb[3];
   "Db_Equipment".Fan[3].IO.DI_OffFeedback := "DB_Simulation".FanOffFb[3];
   "Db_Equipment".Fan[3].IO.DI_Fault := "DB_Simulation".FanFaultFb[3];
END_REGION

REGION Network 12
   RUNG wire#powerrail
      Contact( "DB_Simulation".FanOnFb[4] )
      Coil( "Db_Equipment".Fan[4].IO.DI_OnFeedback )
   END_RUNG
   RUNG wire#powerrail
      Contact( "DB_Simulation".FanOffFb[4] )
      Coil( "Db_Equipment".Fan[4].IO.DI_OffFeedback )
   END_RUNG
   RUNG wire#powerrail
      Contact( "DB_Simulation".FanFaultFb[4] )
      Coil( "Db_Equipment".Fan[4].IO.DI_Fault )
   END_RUNG
   // the same network as SCL:
   "Db_Equipment".Fan[4].IO.DI_OnFeedback := "DB_Simulation".FanOnFb[4];
   "Db_Equipment".Fan[4].IO.DI_OffFeedback := "DB_Simulation".FanOffFb[4];
   "Db_Equipment".Fan[4].IO.DI_Fault := "DB_Simulation".FanFaultFb[4];
END_REGION

REGION Network 13
   RUNG wire#powerrail
      Contact( "DB_Simulation".FanOnFb[5] )
      Coil( "Db_Equipment".Fan[5].IO.DI_OnFeedback )
   END_RUNG
   RUNG wire#powerrail
      Contact( "DB_Simulation".FanOffFb[5] )
      Coil( "Db_Equipment".Fan[5].IO.DI_OffFeedback )
   END_RUNG
   RUNG wire#powerrail
      Contact( "DB_Simulation".FanFaultFb[5] )
      Coil( "Db_Equipment".Fan[5].IO.DI_Fault )
   END_RUNG
   // the same network as SCL:
   "Db_Equipment".Fan[5].IO.DI_OnFeedback := "DB_Simulation".FanOnFb[5];
   "Db_Equipment".Fan[5].IO.DI_OffFeedback := "DB_Simulation".FanOffFb[5];
   "Db_Equipment".Fan[5].IO.DI_Fault := "DB_Simulation".FanFaultFb[5];
END_REGION

REGION Network 14
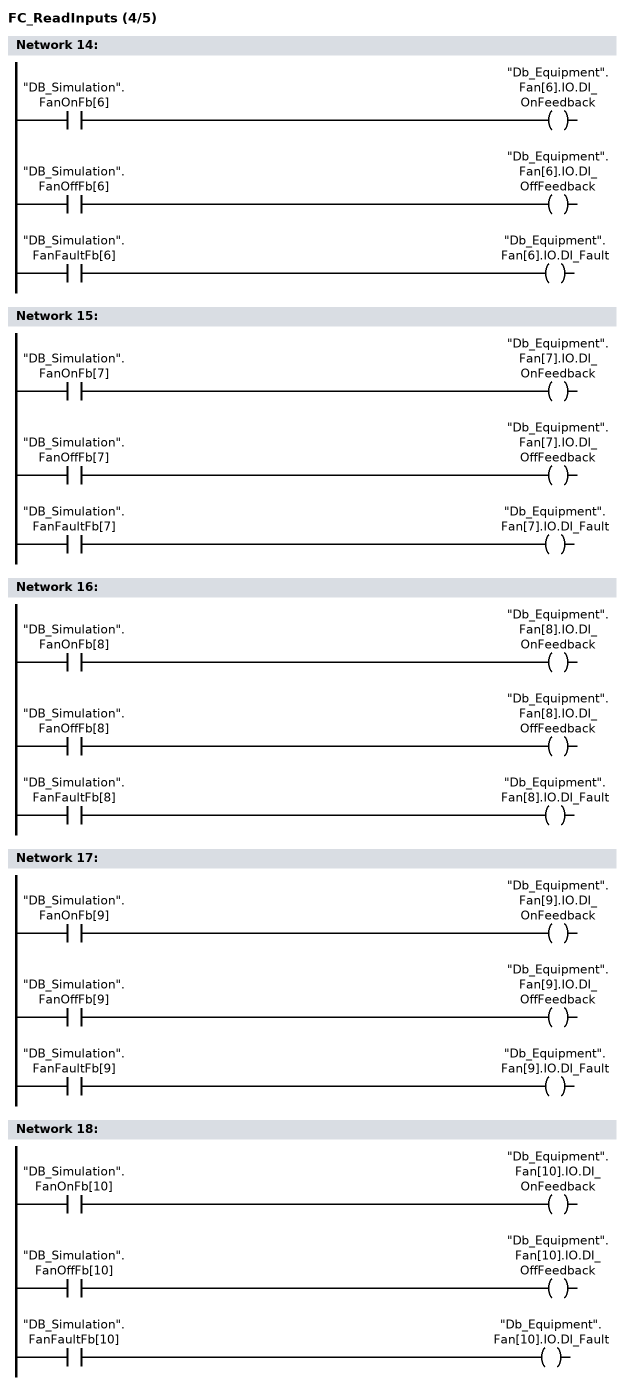
   RUNG wire#powerrail
      Contact( "DB_Simulation".FanOnFb[6] )
      Coil( "Db_Equipment".Fan[6].IO.DI_OnFeedback )
   END_RUNG
   RUNG wire#powerrail
      Contact( "DB_Simulation".FanOffFb[6] )
      Coil( "Db_Equipment".Fan[6].IO.DI_OffFeedback )
   END_RUNG
   RUNG wire#powerrail
      Contact( "DB_Simulation".FanFaultFb[6] )
      Coil( "Db_Equipment".Fan[6].IO.DI_Fault )
   END_RUNG
   // the same network as SCL:
   "Db_Equipment".Fan[6].IO.DI_OnFeedback := "DB_Simulation".FanOnFb[6];
   "Db_Equipment".Fan[6].IO.DI_OffFeedback := "DB_Simulation".FanOffFb[6];
   "Db_Equipment".Fan[6].IO.DI_Fault := "DB_Simulation".FanFaultFb[6];
END_REGION

REGION Network 15
   RUNG wire#powerrail
      Contact( "DB_Simulation".FanOnFb[7] )
      Coil( "Db_Equipment".Fan[7].IO.DI_OnFeedback )
   END_RUNG
   RUNG wire#powerrail
      Contact( "DB_Simulation".FanOffFb[7] )
      Coil( "Db_Equipment".Fan[7].IO.DI_OffFeedback )
   END_RUNG
   RUNG wire#powerrail
      Contact( "DB_Simulation".FanFaultFb[7] )
      Coil( "Db_Equipment".Fan[7].IO.DI_Fault )
   END_RUNG
   // the same network as SCL:
   "Db_Equipment".Fan[7].IO.DI_OnFeedback := "DB_Simulation".FanOnFb[7];
   "Db_Equipment".Fan[7].IO.DI_OffFeedback := "DB_Simulation".FanOffFb[7];
   "Db_Equipment".Fan[7].IO.DI_Fault := "DB_Simulation".FanFaultFb[7];
END_REGION

REGION Network 16
   RUNG wire#powerrail
      Contact( "DB_Simulation".FanOnFb[8] )
      Coil( "Db_Equipment".Fan[8].IO.DI_OnFeedback )
   END_RUNG
   RUNG wire#powerrail
      Contact( "DB_Simulation".FanOffFb[8] )
      Coil( "Db_Equipment".Fan[8].IO.DI_OffFeedback )
   END_RUNG
   RUNG wire#powerrail
      Contact( "DB_Simulation".FanFaultFb[8] )
      Coil( "Db_Equipment".Fan[8].IO.DI_Fault )
   END_RUNG
   // the same network as SCL:
   "Db_Equipment".Fan[8].IO.DI_OnFeedback := "DB_Simulation".FanOnFb[8];
   "Db_Equipment".Fan[8].IO.DI_OffFeedback := "DB_Simulation".FanOffFb[8];
   "Db_Equipment".Fan[8].IO.DI_Fault := "DB_Simulation".FanFaultFb[8];
END_REGION

REGION Network 17
   RUNG wire#powerrail
      Contact( "DB_Simulation".FanOnFb[9] )
      Coil( "Db_Equipment".Fan[9].IO.DI_OnFeedback )
   END_RUNG
   RUNG wire#powerrail
      Contact( "DB_Simulation".FanOffFb[9] )
      Coil( "Db_Equipment".Fan[9].IO.DI_OffFeedback )
   END_RUNG
   RUNG wire#powerrail
      Contact( "DB_Simulation".FanFaultFb[9] )
      Coil( "Db_Equipment".Fan[9].IO.DI_Fault )
   END_RUNG
   // the same network as SCL:
   "Db_Equipment".Fan[9].IO.DI_OnFeedback := "DB_Simulation".FanOnFb[9];
   "Db_Equipment".Fan[9].IO.DI_OffFeedback := "DB_Simulation".FanOffFb[9];
   "Db_Equipment".Fan[9].IO.DI_Fault := "DB_Simulation".FanFaultFb[9];
END_REGION

REGION Network 18
   RUNG wire#powerrail
      Contact( "DB_Simulation".FanOnFb[10] )
      Coil( "Db_Equipment".Fan[10].IO.DI_OnFeedback )
   END_RUNG
   RUNG wire#powerrail
      Contact( "DB_Simulation".FanOffFb[10] )
      Coil( "Db_Equipment".Fan[10].IO.DI_OffFeedback )
   END_RUNG
   RUNG wire#powerrail
      Contact( "DB_Simulation".FanFaultFb[10] )
      Coil( "Db_Equipment".Fan[10].IO.DI_Fault )
   END_RUNG
   // the same network as SCL:
   "Db_Equipment".Fan[10].IO.DI_OnFeedback := "DB_Simulation".FanOnFb[10];
   "Db_Equipment".Fan[10].IO.DI_OffFeedback := "DB_Simulation".FanOffFb[10];
   "Db_Equipment".Fan[10].IO.DI_Fault := "DB_Simulation".FanFaultFb[10];
END_REGION

REGION Network 19
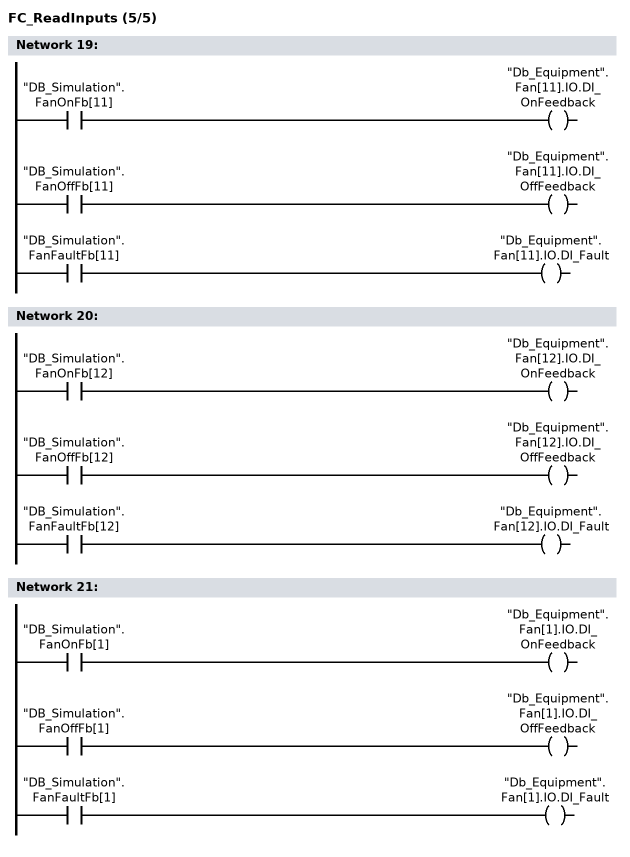
   RUNG wire#powerrail
      Contact( "DB_Simulation".FanOnFb[11] )
      Coil( "Db_Equipment".Fan[11].IO.DI_OnFeedback )
   END_RUNG
   RUNG wire#powerrail
      Contact( "DB_Simulation".FanOffFb[11] )
      Coil( "Db_Equipment".Fan[11].IO.DI_OffFeedback )
   END_RUNG
   RUNG wire#powerrail
      Contact( "DB_Simulation".FanFaultFb[11] )
      Coil( "Db_Equipment".Fan[11].IO.DI_Fault )
   END_RUNG
   // the same network as SCL:
   "Db_Equipment".Fan[11].IO.DI_OnFeedback := "DB_Simulation".FanOnFb[11];
   "Db_Equipment".Fan[11].IO.DI_OffFeedback := "DB_Simulation".FanOffFb[11];
   "Db_Equipment".Fan[11].IO.DI_Fault := "DB_Simulation".FanFaultFb[11];
END_REGION

REGION Network 20
   RUNG wire#powerrail
      Contact( "DB_Simulation".FanOnFb[12] )
      Coil( "Db_Equipment".Fan[12].IO.DI_OnFeedback )
   END_RUNG
   RUNG wire#powerrail
      Contact( "DB_Simulation".FanOffFb[12] )
      Coil( "Db_Equipment".Fan[12].IO.DI_OffFeedback )
   END_RUNG
   RUNG wire#powerrail
      Contact( "DB_Simulation".FanFaultFb[12] )
      Coil( "Db_Equipment".Fan[12].IO.DI_Fault )
   END_RUNG
   // the same network as SCL:
   "Db_Equipment".Fan[12].IO.DI_OnFeedback := "DB_Simulation".FanOnFb[12];
   "Db_Equipment".Fan[12].IO.DI_OffFeedback := "DB_Simulation".FanOffFb[12];
   "Db_Equipment".Fan[12].IO.DI_Fault := "DB_Simulation".FanFaultFb[12];
END_REGION

REGION Network 21
   RUNG wire#powerrail
      Contact( "DB_Simulation".FanOnFb[1] )
      Coil( "Db_Equipment".Fan[1].IO.DI_OnFeedback )
   END_RUNG
   RUNG wire#powerrail
      Contact( "DB_Simulation".FanOffFb[1] )
      Coil( "Db_Equipment".Fan[1].IO.DI_OffFeedback )
   END_RUNG
   RUNG wire#powerrail
      Contact( "DB_Simulation".FanFaultFb[1] )
      Coil( "Db_Equipment".Fan[1].IO.DI_Fault )
   END_RUNG
   // the same network as SCL:
   "Db_Equipment".Fan[1].IO.DI_OnFeedback := "DB_Simulation".FanOnFb[1];
   "Db_Equipment".Fan[1].IO.DI_OffFeedback := "DB_Simulation".FanOffFb[1];
   "Db_Equipment".Fan[1].IO.DI_Fault := "DB_Simulation".FanFaultFb[1];
END_REGION
END_FUNCTION

FUNCTION "FC_WriteOutputs" : Void   // FC3, LAD
{ S7_Optimized_Access := 'TRUE' }
VERSION : 0.1
BEGIN

REGION Network 1
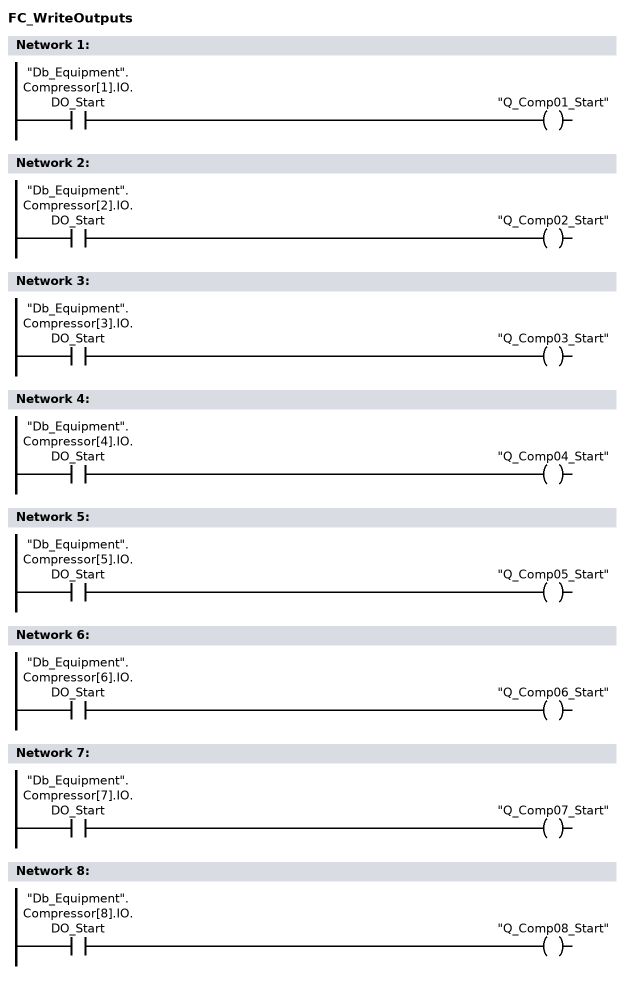
   RUNG wire#powerrail
      Contact( "Db_Equipment".Compressor[1].IO.DO_Start )
      Coil( "Q_Comp01_Start" )
   END_RUNG
   // the same network as SCL:
   "Q_Comp01_Start" := "Db_Equipment".Compressor[1].IO.DO_Start;
END_REGION

REGION Network 2
   RUNG wire#powerrail
      Contact( "Db_Equipment".Compressor[2].IO.DO_Start )
      Coil( "Q_Comp02_Start" )
   END_RUNG
   // the same network as SCL:
   "Q_Comp02_Start" := "Db_Equipment".Compressor[2].IO.DO_Start;
END_REGION

REGION Network 3
   RUNG wire#powerrail
      Contact( "Db_Equipment".Compressor[3].IO.DO_Start )
      Coil( "Q_Comp03_Start" )
   END_RUNG
   // the same network as SCL:
   "Q_Comp03_Start" := "Db_Equipment".Compressor[3].IO.DO_Start;
END_REGION

REGION Network 4
   RUNG wire#powerrail
      Contact( "Db_Equipment".Compressor[4].IO.DO_Start )
      Coil( "Q_Comp04_Start" )
   END_RUNG
   // the same network as SCL:
   "Q_Comp04_Start" := "Db_Equipment".Compressor[4].IO.DO_Start;
END_REGION

REGION Network 5
   RUNG wire#powerrail
      Contact( "Db_Equipment".Compressor[5].IO.DO_Start )
      Coil( "Q_Comp05_Start" )
   END_RUNG
   // the same network as SCL:
   "Q_Comp05_Start" := "Db_Equipment".Compressor[5].IO.DO_Start;
END_REGION

REGION Network 6
   RUNG wire#powerrail
      Contact( "Db_Equipment".Compressor[6].IO.DO_Start )
      Coil( "Q_Comp06_Start" )
   END_RUNG
   // the same network as SCL:
   "Q_Comp06_Start" := "Db_Equipment".Compressor[6].IO.DO_Start;
END_REGION

REGION Network 7
   RUNG wire#powerrail
      Contact( "Db_Equipment".Compressor[7].IO.DO_Start )
      Coil( "Q_Comp07_Start" )
   END_RUNG
   // the same network as SCL:
   "Q_Comp07_Start" := "Db_Equipment".Compressor[7].IO.DO_Start;
END_REGION

REGION Network 8
   RUNG wire#powerrail
      Contact( "Db_Equipment".Compressor[8].IO.DO_Start )
      Coil( "Q_Comp08_Start" )
   END_RUNG
   // the same network as SCL:
   "Q_Comp08_Start" := "Db_Equipment".Compressor[8].IO.DO_Start;
END_REGION
END_FUNCTION

FUNCTION "FC_DemandToCount" : Void   // FC4, LAD
{ S7_Optimized_Access := 'TRUE' }
VERSION : 0.1
   VAR_INPUT
      DemandPercent : Real;
      TotalCount : Int;
   END_VAR
   VAR_OUTPUT
      RequiredCount : Int;
   END_VAR
   VAR_TEMP
      TotalReal : Real;
      ScaleDemand : Real;
      DemandUnits : Real;
   END_VAR
BEGIN

REGION Network 1
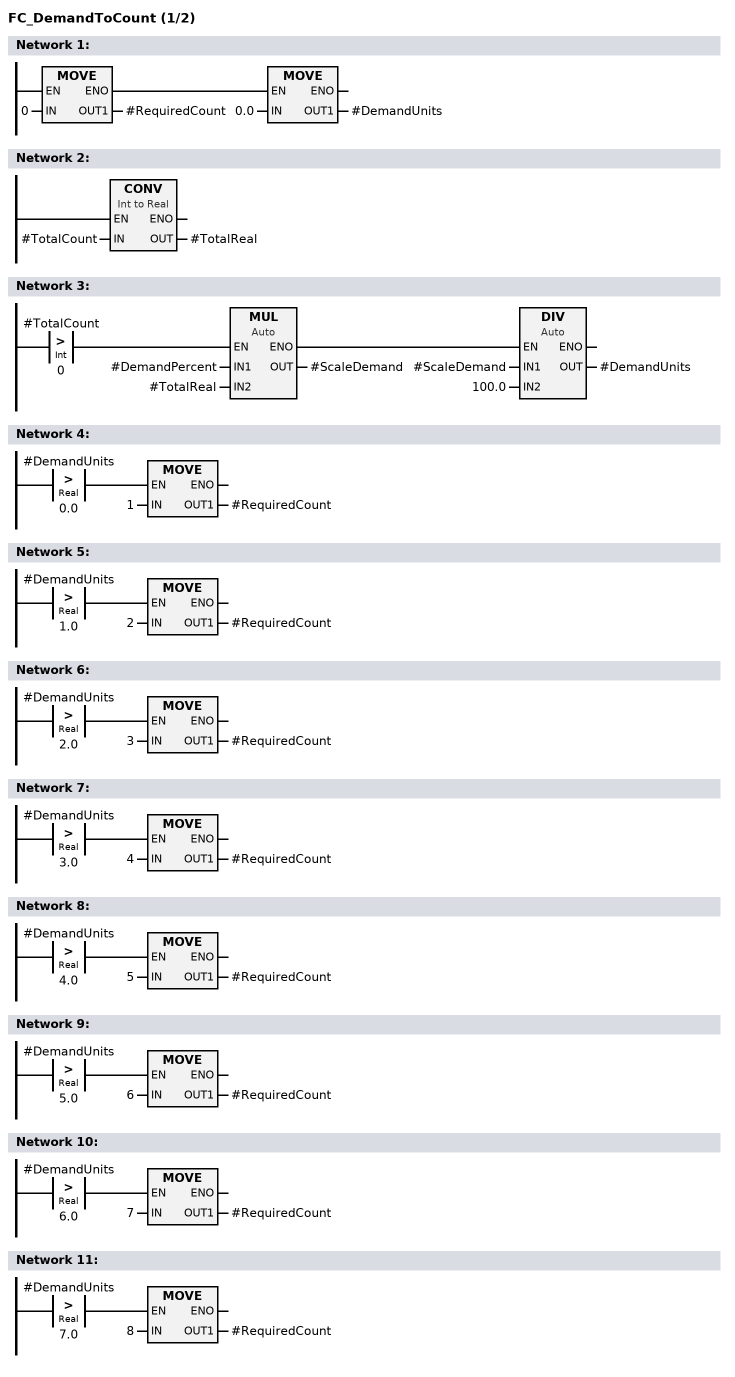
   RUNG wire#powerrail
      Move(in := 0, out1 => #RequiredCount)
      Move(in := 0.0, out1 => #DemandUnits)
   END_RUNG
   // the same network as SCL:
   #RequiredCount := 0;
   #DemandUnits := 0.0;
END_REGION

REGION Network 2
   RUNG wire#powerrail
      { S7_Templates := "[SrcType := Int, DestType := Real]" } Convert(in := #TotalCount, out => #TotalReal)
   END_RUNG
   // the same network as SCL:
   #TotalReal := INT_TO_REAL(#TotalCount);
END_REGION

REGION Network 3
   RUNG wire#powerrail
      { S7_Templates := "SrcType := Int" } GT_Contact(in1 := #TotalCount, in2 := 0)
      Mul(in1 := #DemandPercent, in2 := #TotalReal, out => #ScaleDemand)
      Div(in1 := #ScaleDemand, in2 := 100.0, out => #DemandUnits)
   END_RUNG
   // the same network as SCL:
   IF #TotalCount > 0 THEN
       #ScaleDemand := #DemandPercent * #TotalReal;
       #DemandUnits := #ScaleDemand / 100.0;
   END_IF;
END_REGION

REGION Network 4
   RUNG wire#powerrail
      { S7_Templates := "SrcType := Real" } GT_Contact(in1 := #DemandUnits, in2 := 0.0)
      Move(in := 1, out1 => #RequiredCount)
   END_RUNG
   // the same network as SCL:
   IF #DemandUnits > 0.0 THEN #RequiredCount := 1; END_IF;
END_REGION

REGION Network 5
   RUNG wire#powerrail
      { S7_Templates := "SrcType := Real" } GT_Contact(in1 := #DemandUnits, in2 := 1.0)
      Move(in := 2, out1 => #RequiredCount)
   END_RUNG
   // the same network as SCL:
   IF #DemandUnits > 1.0 THEN #RequiredCount := 2; END_IF;
END_REGION

REGION Network 6
   RUNG wire#powerrail
      { S7_Templates := "SrcType := Real" } GT_Contact(in1 := #DemandUnits, in2 := 2.0)
      Move(in := 3, out1 => #RequiredCount)
   END_RUNG
   // the same network as SCL:
   IF #DemandUnits > 2.0 THEN #RequiredCount := 3; END_IF;
END_REGION

REGION Network 7
   RUNG wire#powerrail
      { S7_Templates := "SrcType := Real" } GT_Contact(in1 := #DemandUnits, in2 := 3.0)
      Move(in := 4, out1 => #RequiredCount)
   END_RUNG
   // the same network as SCL:
   IF #DemandUnits > 3.0 THEN #RequiredCount := 4; END_IF;
END_REGION

REGION Network 8
   RUNG wire#powerrail
      { S7_Templates := "SrcType := Real" } GT_Contact(in1 := #DemandUnits, in2 := 4.0)
      Move(in := 5, out1 => #RequiredCount)
   END_RUNG
   // the same network as SCL:
   IF #DemandUnits > 4.0 THEN #RequiredCount := 5; END_IF;
END_REGION

REGION Network 9
   RUNG wire#powerrail
      { S7_Templates := "SrcType := Real" } GT_Contact(in1 := #DemandUnits, in2 := 5.0)
      Move(in := 6, out1 => #RequiredCount)
   END_RUNG
   // the same network as SCL:
   IF #DemandUnits > 5.0 THEN #RequiredCount := 6; END_IF;
END_REGION

REGION Network 10
   RUNG wire#powerrail
      { S7_Templates := "SrcType := Real" } GT_Contact(in1 := #DemandUnits, in2 := 6.0)
      Move(in := 7, out1 => #RequiredCount)
   END_RUNG
   // the same network as SCL:
   IF #DemandUnits > 6.0 THEN #RequiredCount := 7; END_IF;
END_REGION

REGION Network 11
   RUNG wire#powerrail
      { S7_Templates := "SrcType := Real" } GT_Contact(in1 := #DemandUnits, in2 := 7.0)
      Move(in := 8, out1 => #RequiredCount)
   END_RUNG
   // the same network as SCL:
   IF #DemandUnits > 7.0 THEN #RequiredCount := 8; END_IF;
END_REGION

REGION Network 12
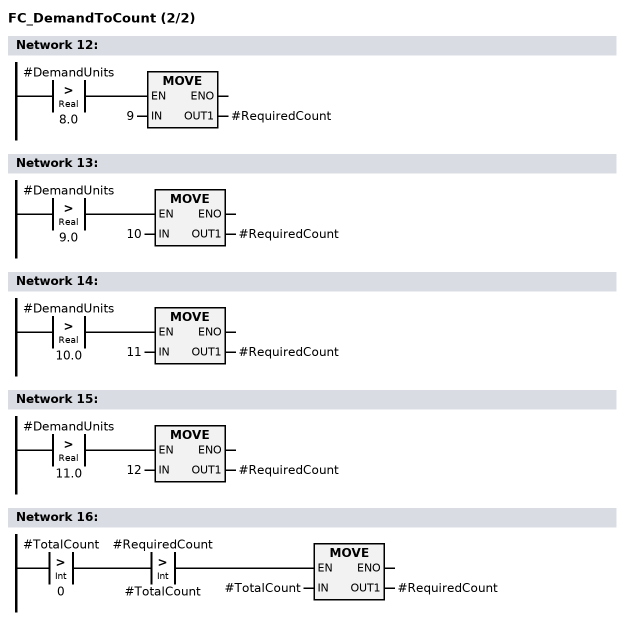
   RUNG wire#powerrail
      { S7_Templates := "SrcType := Real" } GT_Contact(in1 := #DemandUnits, in2 := 8.0)
      Move(in := 9, out1 => #RequiredCount)
   END_RUNG
   // the same network as SCL:
   IF #DemandUnits > 8.0 THEN #RequiredCount := 9; END_IF;
END_REGION

REGION Network 13
   RUNG wire#powerrail
      { S7_Templates := "SrcType := Real" } GT_Contact(in1 := #DemandUnits, in2 := 9.0)
      Move(in := 10, out1 => #RequiredCount)
   END_RUNG
   // the same network as SCL:
   IF #DemandUnits > 9.0 THEN #RequiredCount := 10; END_IF;
END_REGION

REGION Network 14
   RUNG wire#powerrail
      { S7_Templates := "SrcType := Real" } GT_Contact(in1 := #DemandUnits, in2 := 10.0)
      Move(in := 11, out1 => #RequiredCount)
   END_RUNG
   // the same network as SCL:
   IF #DemandUnits > 10.0 THEN #RequiredCount := 11; END_IF;
END_REGION

REGION Network 15
   RUNG wire#powerrail
      { S7_Templates := "SrcType := Real" } GT_Contact(in1 := #DemandUnits, in2 := 11.0)
      Move(in := 12, out1 => #RequiredCount)
   END_RUNG
   // the same network as SCL:
   IF #DemandUnits > 11.0 THEN #RequiredCount := 12; END_IF;
END_REGION

REGION Network 16
   RUNG wire#powerrail
      { S7_Templates := "SrcType := Int" } GT_Contact(in1 := #TotalCount, in2 := 0)
      { S7_Templates := "SrcType := Int" } GT_Contact(in1 := #RequiredCount, in2 := #TotalCount)
      Move(in := #TotalCount, out1 => #RequiredCount)
   END_RUNG
   // the same network as SCL:
   IF (#TotalCount > 0) AND (#RequiredCount > #TotalCount) THEN #RequiredCount := #TotalCount; END_IF;
END_REGION
END_FUNCTION

FUNCTION "FC_AlarmMapping" : Void   // FC5, LAD
{ S7_Optimized_Access := 'TRUE' }
VERSION : 0.1
BEGIN

REGION Network 1
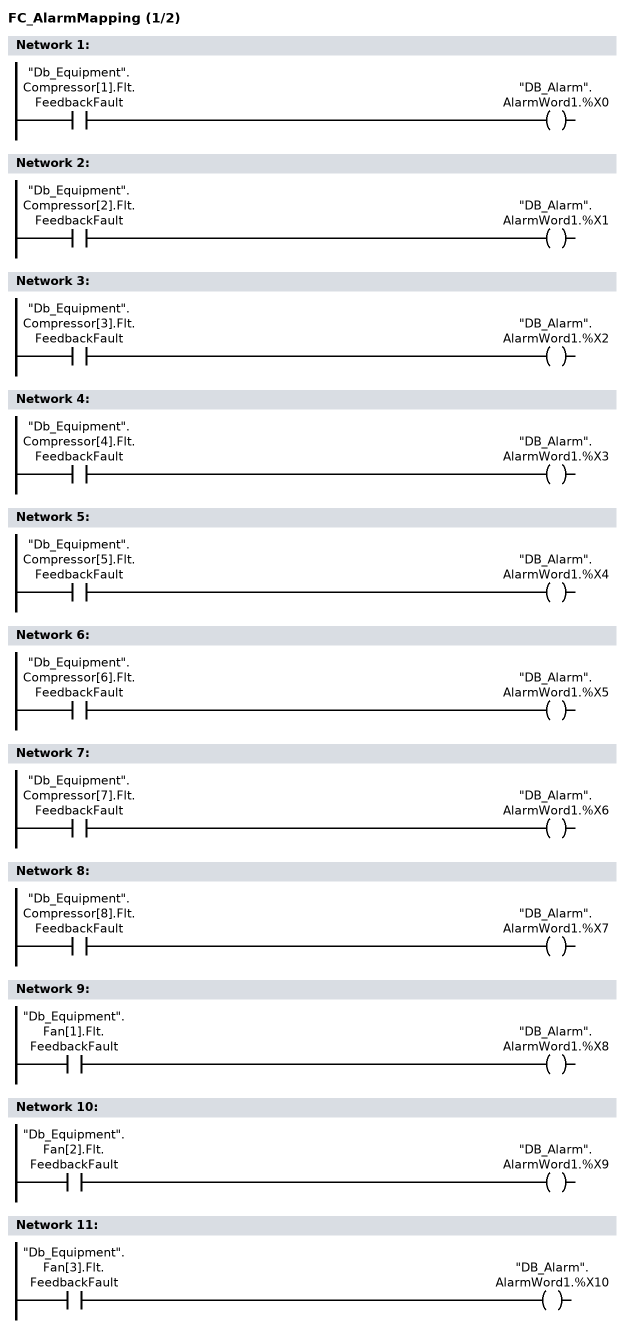
   RUNG wire#powerrail
      Contact( "Db_Equipment".Compressor[1].Flt.FeedbackFault )
      Coil( "DB_Alarm".AlarmWord1.%X0 )
   END_RUNG
   // the same network as SCL:
   "DB_Alarm".AlarmWord1.%X0 := "Db_Equipment".Compressor[1].Flt.FeedbackFault;
END_REGION

REGION Network 2
   RUNG wire#powerrail
      Contact( "Db_Equipment".Compressor[2].Flt.FeedbackFault )
      Coil( "DB_Alarm".AlarmWord1.%X1 )
   END_RUNG
   // the same network as SCL:
   "DB_Alarm".AlarmWord1.%X1 := "Db_Equipment".Compressor[2].Flt.FeedbackFault;
END_REGION

REGION Network 3
   RUNG wire#powerrail
      Contact( "Db_Equipment".Compressor[3].Flt.FeedbackFault )
      Coil( "DB_Alarm".AlarmWord1.%X2 )
   END_RUNG
   // the same network as SCL:
   "DB_Alarm".AlarmWord1.%X2 := "Db_Equipment".Compressor[3].Flt.FeedbackFault;
END_REGION

REGION Network 4
   RUNG wire#powerrail
      Contact( "Db_Equipment".Compressor[4].Flt.FeedbackFault )
      Coil( "DB_Alarm".AlarmWord1.%X3 )
   END_RUNG
   // the same network as SCL:
   "DB_Alarm".AlarmWord1.%X3 := "Db_Equipment".Compressor[4].Flt.FeedbackFault;
END_REGION

REGION Network 5
   RUNG wire#powerrail
      Contact( "Db_Equipment".Compressor[5].Flt.FeedbackFault )
      Coil( "DB_Alarm".AlarmWord1.%X4 )
   END_RUNG
   // the same network as SCL:
   "DB_Alarm".AlarmWord1.%X4 := "Db_Equipment".Compressor[5].Flt.FeedbackFault;
END_REGION

REGION Network 6
   RUNG wire#powerrail
      Contact( "Db_Equipment".Compressor[6].Flt.FeedbackFault )
      Coil( "DB_Alarm".AlarmWord1.%X5 )
   END_RUNG
   // the same network as SCL:
   "DB_Alarm".AlarmWord1.%X5 := "Db_Equipment".Compressor[6].Flt.FeedbackFault;
END_REGION

REGION Network 7
   RUNG wire#powerrail
      Contact( "Db_Equipment".Compressor[7].Flt.FeedbackFault )
      Coil( "DB_Alarm".AlarmWord1.%X6 )
   END_RUNG
   // the same network as SCL:
   "DB_Alarm".AlarmWord1.%X6 := "Db_Equipment".Compressor[7].Flt.FeedbackFault;
END_REGION

REGION Network 8
   RUNG wire#powerrail
      Contact( "Db_Equipment".Compressor[8].Flt.FeedbackFault )
      Coil( "DB_Alarm".AlarmWord1.%X7 )
   END_RUNG
   // the same network as SCL:
   "DB_Alarm".AlarmWord1.%X7 := "Db_Equipment".Compressor[8].Flt.FeedbackFault;
END_REGION

REGION Network 9
   RUNG wire#powerrail
      Contact( "Db_Equipment".Fan[1].Flt.FeedbackFault )
      Coil( "DB_Alarm".AlarmWord1.%X8 )
   END_RUNG
   // the same network as SCL:
   "DB_Alarm".AlarmWord1.%X8 := "Db_Equipment".Fan[1].Flt.FeedbackFault;
END_REGION

REGION Network 10
   RUNG wire#powerrail
      Contact( "Db_Equipment".Fan[2].Flt.FeedbackFault )
      Coil( "DB_Alarm".AlarmWord1.%X9 )
   END_RUNG
   // the same network as SCL:
   "DB_Alarm".AlarmWord1.%X9 := "Db_Equipment".Fan[2].Flt.FeedbackFault;
END_REGION

REGION Network 11
   RUNG wire#powerrail
      Contact( "Db_Equipment".Fan[3].Flt.FeedbackFault )
      Coil( "DB_Alarm".AlarmWord1.%X10 )
   END_RUNG
   // the same network as SCL:
   "DB_Alarm".AlarmWord1.%X10 := "Db_Equipment".Fan[3].Flt.FeedbackFault;
END_REGION

REGION Network 12
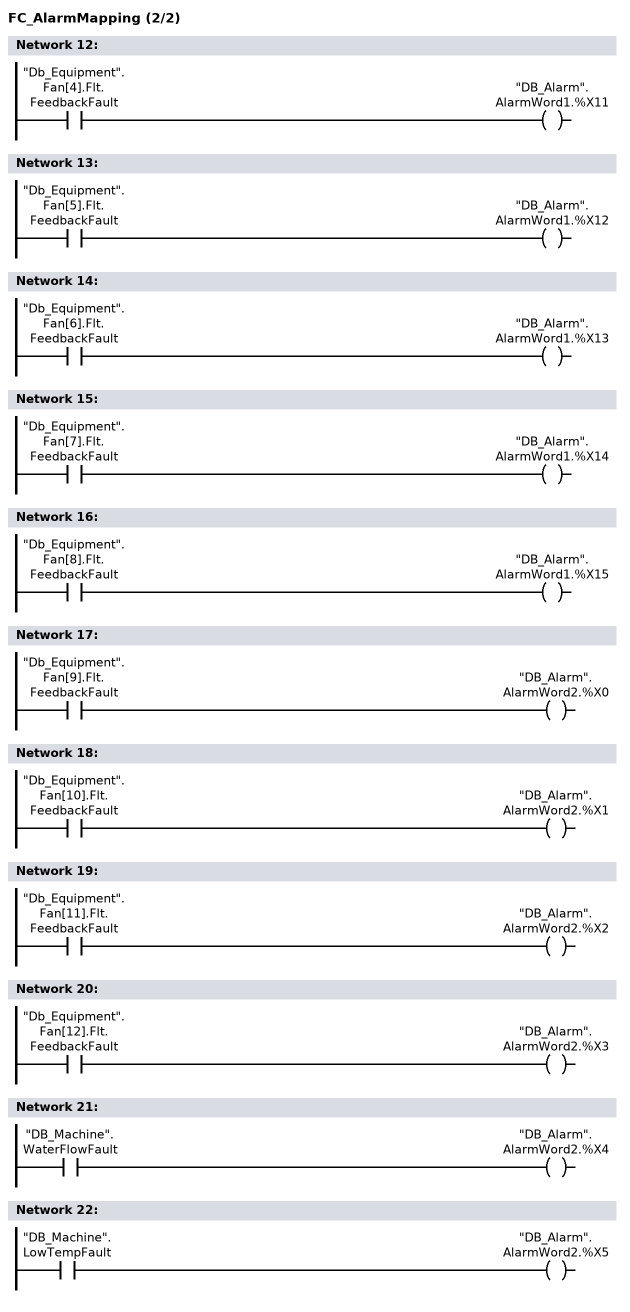
   RUNG wire#powerrail
      Contact( "Db_Equipment".Fan[4].Flt.FeedbackFault )
      Coil( "DB_Alarm".AlarmWord1.%X11 )
   END_RUNG
   // the same network as SCL:
   "DB_Alarm".AlarmWord1.%X11 := "Db_Equipment".Fan[4].Flt.FeedbackFault;
END_REGION

REGION Network 13
   RUNG wire#powerrail
      Contact( "Db_Equipment".Fan[5].Flt.FeedbackFault )
      Coil( "DB_Alarm".AlarmWord1.%X12 )
   END_RUNG
   // the same network as SCL:
   "DB_Alarm".AlarmWord1.%X12 := "Db_Equipment".Fan[5].Flt.FeedbackFault;
END_REGION

REGION Network 14
   RUNG wire#powerrail
      Contact( "Db_Equipment".Fan[6].Flt.FeedbackFault )
      Coil( "DB_Alarm".AlarmWord1.%X13 )
   END_RUNG
   // the same network as SCL:
   "DB_Alarm".AlarmWord1.%X13 := "Db_Equipment".Fan[6].Flt.FeedbackFault;
END_REGION

REGION Network 15
   RUNG wire#powerrail
      Contact( "Db_Equipment".Fan[7].Flt.FeedbackFault )
      Coil( "DB_Alarm".AlarmWord1.%X14 )
   END_RUNG
   // the same network as SCL:
   "DB_Alarm".AlarmWord1.%X14 := "Db_Equipment".Fan[7].Flt.FeedbackFault;
END_REGION

REGION Network 16
   RUNG wire#powerrail
      Contact( "Db_Equipment".Fan[8].Flt.FeedbackFault )
      Coil( "DB_Alarm".AlarmWord1.%X15 )
   END_RUNG
   // the same network as SCL:
   "DB_Alarm".AlarmWord1.%X15 := "Db_Equipment".Fan[8].Flt.FeedbackFault;
END_REGION

REGION Network 17
   RUNG wire#powerrail
      Contact( "Db_Equipment".Fan[9].Flt.FeedbackFault )
      Coil( "DB_Alarm".AlarmWord2.%X0 )
   END_RUNG
   // the same network as SCL:
   "DB_Alarm".AlarmWord2.%X0 := "Db_Equipment".Fan[9].Flt.FeedbackFault;
END_REGION

REGION Network 18
   RUNG wire#powerrail
      Contact( "Db_Equipment".Fan[10].Flt.FeedbackFault )
      Coil( "DB_Alarm".AlarmWord2.%X1 )
   END_RUNG
   // the same network as SCL:
   "DB_Alarm".AlarmWord2.%X1 := "Db_Equipment".Fan[10].Flt.FeedbackFault;
END_REGION

REGION Network 19
   RUNG wire#powerrail
      Contact( "Db_Equipment".Fan[11].Flt.FeedbackFault )
      Coil( "DB_Alarm".AlarmWord2.%X2 )
   END_RUNG
   // the same network as SCL:
   "DB_Alarm".AlarmWord2.%X2 := "Db_Equipment".Fan[11].Flt.FeedbackFault;
END_REGION

REGION Network 20
   RUNG wire#powerrail
      Contact( "Db_Equipment".Fan[12].Flt.FeedbackFault )
      Coil( "DB_Alarm".AlarmWord2.%X3 )
   END_RUNG
   // the same network as SCL:
   "DB_Alarm".AlarmWord2.%X3 := "Db_Equipment".Fan[12].Flt.FeedbackFault;
END_REGION

REGION Network 21
   RUNG wire#powerrail
      Contact( "DB_Machine".WaterFlowFault )
      Coil( "DB_Alarm".AlarmWord2.%X4 )
   END_RUNG
   // the same network as SCL:
   "DB_Alarm".AlarmWord2.%X4 := "DB_Machine".WaterFlowFault;
END_REGION

REGION Network 22
   RUNG wire#powerrail
      Contact( "DB_Machine".LowTempFault )
      Coil( "DB_Alarm".AlarmWord2.%X5 )
   END_RUNG
   // the same network as SCL:
   "DB_Alarm".AlarmWord2.%X5 := "DB_Machine".LowTempFault;
END_REGION
END_FUNCTION

// folder: 04_similation

FUNCTION_BLOCK "FB_CompressorSim"   // FB7, LAD
{ S7_Optimized_Access := 'TRUE' }
VERSION : 0.1
   VAR_INPUT
      StartCommand : Bool;
   END_VAR
   VAR_OUTPUT
      OnFeedBack : Bool;
      OffFeedback : Bool;
   END_VAR
   VAR
      tStopDelay : Bool;
      tStartDelay : TON_TIME;
   END_VAR
BEGIN

REGION Network 1
